# B&R Automation Studio project A2019059_Linka_Power_CP (part 33)

```iecst
            IF P2_StoperZvarania.IN.Centrovanie_ZASUNUTE_IS17 THEN
                SC_P2_StoperZvarania.ResetStep:= TRUE;
                SC_P2_StoperZvarania.Step:= 550;
            END_IF

            //Odoslanie dát na server//

        550:
            SC_P2_StoperZvarania.StepName:='550 - Automaticky Rezim - odoslanie stavu paletky na server';
            SC_P2_StoperZvarania.IdleTime.PT:= T#200ms;
            SC_P2_StoperZvarania.AlarmTime.PT:= T#5s;

            IF NOT SC_P2_StoperZvarania.Switch1 THEN
                TRCB_P2_Zvaranie_ST6.CMD.OdosliStavPaletky_TYP2:= TRUE;
                SC_P2_StoperZvarania.Switch1:= TRUE;
            END_IF

            IF TRCB_P2_Zvaranie_ST6.STATUS.KomunikaciaUkoncena THEN
                TRCB_P2_Zvaranie_ST6.CMD.OdosliStavPaletky_TYP2:= FALSE;
                SC_P2_StoperZvarania.ResetStep:= TRUE;
                SC_P2_StoperZvarania.Step:= 553;
            ELSIF TRCB_P2_Zvaranie_ST6.STATUS.KomunikaciaError THEN
                //                P2_Alarmy[236]:= TRUE;
                //                P2_PoruchaST4:= TRUE;
            END_IF

        553:
            SC_P2_StoperZvarania.StepName:='553 - Automaticky Rezim - kontrola odpovede servera';
            SC_P2_StoperZvarania.IdleTime.PT:= T#200ms;
            SC_P2_StoperZvarania.AlarmTime.PT:= T#5s;

            IF NOT TRCB_P2_Zvaranie_ST6.STATUS.KomunikaciaUkoncena THEN
                IF TRCB_P2_Zvaranie_ST6.OUTPUTS.PovolenieCinnostiNaPaletke = 'OK' THEN
                    SC_P2_StoperZvarania.ResetStep:= TRUE;
                    SC_P2_StoperZvarania.Step:= 555;
                ELSIF TRCB_P2_Zvaranie_ST6.OUTPUTS.PovolenieCinnostiNaPaletke = 'NG' THEN
                    Paletka[i].PAR.StavPaletky:= 'NG';
                    SC_P2_StoperZvarania.ResetStep:= TRUE;
                    SC_P2_StoperZvarania.Step:= 555;
                END_IF
            END_IF

        555:
            SC_P2_StoperZvarania.StepName:='555 - Automaticky Rezim - vyhodnotenie stavu paletky';
            SC_P2_StoperZvarania.IdleTime.PT:= T#200ms;
            SC_P2_StoperZvarania.AlarmTime.PT:= T#10s;

            IF Paletka[i].PAR.StavPaletky = 'OK' THEN
                IF Paletka[i].PAR.StavPowerCP = 'PASS' THEN
                    Paletka[i].PAR.StavPaletky:= 'OK';
                ELSIF Paletka[i].PAR.StavPowerCP = 'FAIL' THEN
                    Paletka[i].PAR.StavPaletky:= 'NG';
                END_IF
            END_IF
            Paletka[i].VnutornyStav.KomunikaciaUzavreta:= TRUE;
            SC_P2_StoperZvarania.ResetStep:= TRUE;
            SC_P2_StoperZvarania.Step:= 560;

            //Vyvezenie paletky//

        560:
            SC_P2_StoperZvarania.StepName:='560 - Automaticky Rezim - cakam na vyvezenie na vstupny stoper bunky 3';
            SC_P2_StoperZvarania.IdleTime.PT:= T#200ms;
            SC_P2_StoperZvarania.AlarmTime.PT:= T#5s;

            IF P2_StoperZvarania.KoniecCyklu THEN
                SC_P2_StoperZvarania.ResetStep:= TRUE;
                SC_P2_StoperZvarania.Step:= 0;
            ELSIF ((NOT P3_VstupnyStoper.IN.PritomnPaletky_IS85 AND SC_P3_VstupnyStoper.Step = 100) OR (P3_VstupnyStoper.OUT.ZasunStoper_YV193 AND SC_P3_VstupnyStoper.Step = 105)) AND NOT P2_StoperZvarania.STAV.PrebiehaVyvezeniePaletky AND NOT TEST THEN
                P2_StoperZvarania.OUT.ZasunStoper_YV59:= TRUE;
                P2_StoperZvarania.STAV.PrebiehaVyvezeniePaletky:= TRUE;
                SC_P2_StoperZvarania.ResetStep:= TRUE;
                SC_P2_StoperZvarania.Step:= 561;
            END_IF

        561:
            SC_P2_StoperZvarania.StepName:='561 - Automaticky Rezim - ukoncenie vyvazania na vstupny stoper bunky 3';
            SC_P2_StoperZvarania.IdleTime.PT:= T#200ms;
            SC_P2_StoperZvarania.AlarmTime.PT:= T#10s;

            SC_P2_StoperZvarania.AlarmTime.IN:= P2_StoperZvarania.IN.PritomnostPaletky_S9;
            SC_P2_StoperZvarania.IdleTime.IN:= NOT P2_StoperZvarania.IN.PritomnostPaletky_S9;

            IF NOT P2_StoperZvarania.IN.PritomnostPaletky_S9 THEN
                IF Revork THEN
                    Paletka[i].PAR.RevorkovyKus:= FALSE;
                    Paletka[i].PAR.CisloRevorkovejStanice:= '';
                    Revork:= FALSE;
                END_IF
                TestovaciKus:= FALSE;
                CisloFotky:= 0;
                Paletka[i].PAR.StavPowerCP:= '';
                Paletka[i].VnutornyStav.CinnostSpustena:= FALSE;
                Paletka[i].VnutornyStav.CinnostUkoncena:= FALSE;
                Paletka[i].VnutornyStav.FotkyOdoslane:= FALSE;
                Paletka[i].VnutornyStav.KomunikaciaOtvorena:= FALSE;
                Paletka[i].VnutornyStav.KomunikaciaUzavreta:= FALSE;
                Reports.Zvaranie.Moment.LavyZvar:= '';
                Reports.Zvaranie.VyslednyReport:= '';
                Reports.Zvaranie.Vyska.LavyZvar:= '';
                Reports.Zvaranie.Frekvencia:= '';
                Reports.Zvaranie.Moment.PravyZvar:= '';
                Reports.Zvaranie.Vyska.PravyZvar:= '';
                Reports.Kamery.P2_CAM11_KontrolaZvaru:= '';
                Reports.Kamery.P2_CAM11_KontrolaPowerCP:= '';
            END_IF

            IF SC_P2_StoperZvarania.IdleTime.Q THEN
                P2_StoperZvarania.OUT.ZasunStoper_YV59:= FALSE;
                SC_P2_StoperZvarania.ResetStep:= TRUE;
                SC_P2_StoperZvarania.Step:= 100;
            ELSIF SC_P2_StoperZvarania.AlarmTime.Q THEN
                P2_Alarmy[289]:= TRUE;
                P2_Pracovisko.KoniecCyklu:= TRUE;
                SC_P2_StoperZvarania.ResetStep:= TRUE;
                SC_P2_StoperZvarania.Step:= 0;
            END_IF

            //*******************************************************Manuálny režim*******************************************************************************//

        700:
            SC_P2_StoperZvarania.StepName:='700 - Manualny Rezim';
            SC_P2_StoperZvarania.IdleTime.PT:= T#8s;
            SC_P2_StoperZvarania.AlarmTime.PT:= T#5s;

    END_CASE

                END_PROGRAM

PROGRAM _EXIT
                (* Insert code here *)

                END_PROGRAM
```

#### Variables.var - Local variables
```iecst
VAR
	SC_OvlCentrovacky : SequenceControlTyp;
	Centrovacku_VYSUN : BOOL;
	Centrovacku_ZASUN : BOOL;
	PrecitaneCisloPaletky : STRING[3];
	ServerOdpoved_StavPowerCP : STRING[5];
	i : USINT;
	TEST : BOOL;
	PocetDopytovNaServer : USINT;
	TestovaciKus : BOOL;
	Revork : BOOL;
	Triger_0 : BOOL;
	Triger_1 : BOOL;
	CisloFotky : USINT;
	PocetZopakovaniOdobratia : USINT;
	PocetTrigrovKamery : USINT;
END_VAR
```

#### OvlCentrovacky.st
```iecst
ACTION OvlCentrovacky:

	//Volanie funkcie SequenceControl//
	SequenceControl(SC:= SC_OvlCentrovacky);

	CASE SC_OvlCentrovacky.Step OF

		0:
			SC_OvlCentrovacky.StepName:= '0 - Nulovanie';
			Centrovacku_VYSUN:= FALSE;
			Centrovacku_ZASUN:= FALSE;
//			P2_StoperZvarania.OUT.VysunCentrovanie_YV60:= FALSE;
//			P2_StoperZvarania.OUT.ZasunCentrovanie_YV61:= FALSE;

			IF SC_P2_StoperZvarania.Step <> 0 THEN
				SC_OvlCentrovacky.ResetStep:= TRUE;
				SC_OvlCentrovacky.Step:= 1;
			END_IF

		1:
			SC_OvlCentrovacky.StepName:= '1 - Rozhodnutie o cinnosti';
			IF Centrovacku_VYSUN THEN
				SC_OvlCentrovacky.Step:= 10;
			ELSIF Centrovacku_ZASUN THEN
				SC_OvlCentrovacky.Step:= 20;
			END_IF

		10:
			SC_OvlCentrovacky.StepName:= '10 - Vysunutie centrovacky';
			SC_OvlCentrovacky.IdleTime.PT:= T#3s;
			SC_OvlCentrovacky.AlarmTime.PT:= T#3s;

			IF P2_StoperZvarania.Automat THEN
				SC_OvlCentrovacky.AlarmTime.IN:= TRUE;
			ELSE
				SC_OvlCentrovacky.IdleTime.IN:= TRUE;
			END_IF

			IF NOT SC_OvlCentrovacky.Switch1 THEN
				P2_StoperZvarania.OUT.ZasunCentrovanie_YV61:= FALSE;
                P2_StoperZvarania.OUT.VysunCentrovanie_YV60:= TRUE;
				SC_OvlCentrovacky.Switch1:= TRUE;
			END_IF

			IF P2_StoperZvarania.IN.Centrovanie_VYSUNUTE_IS16 OR SC_OvlCentrovacky.IdleTime.Q THEN
				SC_OvlCentrovacky.ResetStep:= TRUE;
				SC_OvlCentrovacky.Step:= 0;
			ELSIF SC_OvlCentrovacky.AlarmTime.Q THEN
				P2_Alarmy[217]:= TRUE;
				P2_PoruchaST4:= TRUE;
			END_IF

		20:
			SC_OvlCentrovacky.StepName:= '20 - Zasunutie centrovacky';
			SC_OvlCentrovacky.IdleTime.PT:= T#3s;
			SC_OvlCentrovacky.AlarmTime.PT:= T#3s;

			IF P2_StoperZvarania.Automat THEN
				SC_OvlCentrovacky.AlarmTime.IN:= TRUE;
			ELSE
				SC_OvlCentrovacky.IdleTime.IN:= TRUE;
			END_IF

			IF NOT SC_OvlCentrovacky.Switch1 THEN
				P2_StoperZvarania.OUT.VysunCentrovanie_YV60:= FALSE;
                P2_StoperZvarania.OUT.ZasunCentrovanie_YV61:= TRUE;
				SC_OvlCentrovacky.Switch1:= TRUE;
			END_IF

			IF P2_StoperZvarania.IN.Centrovanie_ZASUNUTE_IS17 OR SC_OvlCentrovacky.IdleTime.Q THEN
				SC_OvlCentrovacky.ResetStep:= TRUE;
				SC_OvlCentrovacky.Step:= 0;
			ELSIF SC_OvlCentrovacky.AlarmTime.Q THEN
				P2_Alarmy[218]:= TRUE;
				P2_PoruchaST4:= TRUE;
			END_IF

	END_CASE

END_ACTION
```

#### StratoveSekundy.st
```iecst
ACTION StratoveSekundy:

END_ACTION
```

#### IOLinkKomunikacia.st
```iecst
ACTION IOLinkKomunikacia:

	//Snímač paletky//
	P2_StoperZvarania.IN.PritomnostPaletky_S9:= P2_StoperZvarania.PAR.SnimacPaletky_IOLinkInputs[1].0;
	P2_StoperZvarania.IN.PrecitaneCisloPaletky_S9:= P2_StoperZvarania.PAR.SnimacPaletky_IOLinkInputs[9];

END_ACTION
```

### Program Logical/Program/Pracovisko_2/P2_Zvaranie (IEC)

#### Main.st - Init, cyclic, exit code
```iecst
PROGRAM _INIT
    P2_Zvaranie.PAR.ServoZdvihu_JoggRychlost:= 5;

    //Zápis do ParID serva - nastavenie max momentu v smere otáčania a v protismere otáčania//
//    NovaHodnotaMomentu_POS := 1.5; //v Nm
//    NovaHodnotaMomentu_NEG := 1.5; //v Nm
//    MC_BR_ProcessParID_AcpAx_0.Axis:= ADR(gAxis_5);
//    MC_BR_ProcessParID_AcpAx_0.DataAddress:= ADR(McAcpAxProcessParIDType_0);
//    MC_BR_ProcessParID_AcpAx_0.NumberOfParIDs:= 2;
//    MC_BR_ProcessParID_AcpAx_0.Mode:= mcACPAX_PARID_SET;
//
//    McAcpAxProcessParIDType_0[0].DataType   := mcACPAX_PARTYPE_REAL;
//    McAcpAxProcessParIDType_0[0].ParID      := 248;
//    McAcpAxProcessParIDType_0[0].VariableAddress    := ADR(NovaHodnotaMomentu_POS);
//
//    McAcpAxProcessParIDType_0[1].DataType   := mcACPAX_PARTYPE_REAL;
//    McAcpAxProcessParIDType_0[1].ParID      := 249;
//    McAcpAxProcessParIDType_0[1].VariableAddress    := ADR(NovaHodnotaMomentu_NEG);
//
//    MC_BR_ProcessParID_AcpAx_0.Execute:= TRUE;
//    MC_BR_ProcessParID_AcpAx_0();

END_PROGRAM

PROGRAM _CYCLIC

     //Index paletky//
    i:= P2_StoperZvarania.PAR.IndexPaletky;

    //Volanie funkcie SequenceControl//
    SequenceControl(SC:= SC_P2_Zvaranie);

    //Volanie podprogramov//
    OvlServaZdvihu;
    OvlPojazdu;

    //Reset sekcie //
    IF NOT Safety.STAV.P2_ZonaBunky_AKTIVNA THEN
        SC_P2_Zvaranie.Step:= 0;
    ELSIF P2_Zvaranie.Reset THEN
        SC_P2_Zvaranie.Step:= 0;
        P2_Zvaranie.Reset:= FALSE;
    END_IF

    //Zastavenie serva//
    IF EDGEPOS(P2_PoruchaST4) THEN
        Zdvih_STOP:= TRUE;
    ELSIF EDGEPOS(P2_Zvaranie.Reset) THEN
        Zdvih_STOP:= TRUE;
    END_IF

    CASE SC_P2_Zvaranie.Step OF

        0:
            SC_P2_Zvaranie.StepName:='0 - Nulovanie';
            SC_OvlZdvihu.Step:= 0;
            P2_Zvaranie.Automat:= FALSE;
            P2_Zvaranie.KoniecCyklu:= FALSE;
            P2_Zvaranie.Manual:= FALSE;
            P2_Zvaranie.STAV.PoINIT:= FALSE;
            P2_Zvaranie.ServoZdvihuZvarania_M6.CMD.JoggLimit_ACTIVE:= FALSE;
            P2_Robot.KOM_OUT.Zvaranie_BezpecnaPozicia:= FALSE;
            P2_Zvaranie.STAV.ServoZdvihu_PoziciaDosiahnuta:= FALSE;
            P2_Zvaranie.OUT.Zvaracka_RESET:= FALSE;
            P2_Zvaranie.OUT.Zvaracka_START:= FALSE;

            IF Safety.STAV.P2_ZonaBunky_AKTIVNA AND NOT P2_Pracovisko.STAV.PORUCHA AND P2_Pracovisko.IN.PrivodVzduchu_SnimacTlaku_S3 AND P2_Pracovisko.STAV.ServaBunky_READY THEN
                SC_P2_Zvaranie.ResetStep:= TRUE;
                SC_P2_Zvaranie.Step:= 1;
            END_IF

        1:
            SC_P2_Zvaranie.StepName:='1 - Cakam na spustenie vyroby';
            P2_Zvaranie.KoniecCyklu:= FALSE;
            IF P2_Zvaranie.Automat THEN
                SC_P2_Zvaranie.Step:= 2;
            ELSIF P2_Zvaranie.Manual THEN
                SC_P2_Zvaranie.Step:= 700;
            END_IF

            //********************************************************Inicializácia****************************************************************************//

        2:
            SC_P2_Zvaranie.StepName:='2 - Inicializacia - cakam na spustenie inicializacie';
            SC_P2_Zvaranie.IdleTime.PT:= T#2s;
            SC_P2_Zvaranie.AlarmTime.PT:= T#5s;

            SC_P2_Zvaranie.IdleTime.IN:= TRUE;

            IF SC_P2_Zvaranie.IdleTime.Q THEN
                SC_P2_Zvaranie.ResetStep:= TRUE;
                SC_P2_Zvaranie.Step:= 3;
            END_IF

        3:
            SC_P2_Zvaranie.StepName:='3 - Inicializacia - kontrola homingu serva zdvihu zvarania';
            SC_P2_Zvaranie.IdleTime.PT:= T#2s;
            SC_P2_Zvaranie.AlarmTime.PT:= T#5s;

            IF P2_Zvaranie.STAV.ServoZdvihu_HomingOK THEN
                SC_P2_Zvaranie.ResetStep:= TRUE;
                SC_P2_Zvaranie.Step:= 5;
            ELSE
                SC_P2_Zvaranie.ResetStep:= TRUE;
                SC_P2_Zvaranie.Step:= 4;
            END_IF

        4:
            SC_P2_Zvaranie.StepName:='4 - Inicializacia - spustenie homingu serva zdvihu zvarania';
            SC_P2_Zvaranie.IdleTime.PT:= T#2s;
            SC_P2_Zvaranie.AlarmTime.PT:= T#5s;

            IF NOT SC_P2_Zvaranie.Switch1 AND Safety.STAV.P2_ZonaBunky_AKTIVNA THEN
                Zdvih_HOME:= TRUE;
                SC_P2_Zvaranie.Switch1:= TRUE;
            END_IF

            IF P2_Zvaranie.STAV.ServoZdvihu_HomingOK THEN
                SC_P2_Zvaranie.ResetStep:= TRUE;
                SC_P2_Zvaranie.Step:= 5;
            END_IF

        5:
            SC_P2_Zvaranie.StepName:='5 - Inicializacia - presun zdvihu zvarania do vychodiskovej pozicie';
            SC_P2_Zvaranie.IdleTime.PT:= T#2s;
            SC_P2_Zvaranie.AlarmTime.PT:= T#5s;

            P2_Zvaranie.PAR.ServoZdvihu_ZadanaPozicia:= 0;

            P2_Robot.KOM_OUT.Zvaranie_BezpecnaPozicia:= FALSE;

            IF NOT SC_P2_Zvaranie.Switch1 AND SC_OvlZdvihu.Step = 1 AND Safety.STAV.P2_ZonaBunky_AKTIVNA THEN
                Zdvih_POLOHUJ:= TRUE;
                SC_P2_Zvaranie.Switch1:= TRUE;
            END_IF

            IF P2_Zvaranie.STAV.ServoZdvihu_PoziciaDosiahnuta THEN
                P2_Zvaranie.STAV.ServoZdvihu_PoziciaDosiahnuta:= FALSE;
                SC_P2_Zvaranie.ResetStep:= TRUE;
                SC_P2_Zvaranie.Step:= 10;
            END_IF

        10:
            SC_P2_Zvaranie.StepName:='10 - Inicializacia - presun pojazdu zvarania vpravo';
            SC_P2_Zvaranie.IdleTime.PT:= T#2s;
            SC_P2_Zvaranie.AlarmTime.PT:= T#5s;

            IF NOT SC_P2_Zvaranie.Switch1 THEN
                PresunVPRAVO:= TRUE;
                SC_P2_Zvaranie.Switch1:= TRUE;
            END_IF

            IF P2_Zvaranie.IN.PojazdZvarania_PozVPRAVO_IS10 THEN
                P2_Robot.KOM_OUT.Zvaranie_BezpecnaPozicia:= TRUE;
                SC_P2_Zvaranie.ResetStep:= TRUE;
                SC_P2_Zvaranie.Step:= 12;
            END_IF

        12:
            SC_P2_Zvaranie.StepName:='12 - Inicializacia - kontrola stavu zvaracky';
            SC_P2_Zvaranie.IdleTime.PT:= T#2s;
            SC_P2_Zvaranie.AlarmTime.PT:= T#5s;

            IF NOT P2_Zvaranie.IN.ZvarackaStav_READY THEN
                SC_P2_Zvaranie.ResetStep:= TRUE;
                SC_P2_Zvaranie.Step:= 15;
            ELSE
                P2_Zvaranie.STAV.PoINIT:= TRUE;
                SC_P2_Zvaranie.ResetStep:= TRUE;
                SC_P2_Zvaranie.Step:= 100;
            END_IF

        15:
            SC_P2_Zvaranie.StepName:='15 - Inicializacia - reset zvaracky';
            SC_P2_Zvaranie.IdleTime.PT:= T#200ms;
            SC_P2_Zvaranie.AlarmTime.PT:= T#5s;

            IF NOT SC_P2_Zvaranie.Switch1 THEN
                P2_Zvaranie.OUT.Zvaracka_RESET:= TRUE;
                SC_P2_Zvaranie.IdleTime.IN:= TRUE;
                SC_P2_Zvaranie.Switch1:= TRUE;
            END_IF

            IF SC_P2_Zvaranie.IdleTime.Q THEN
                P2_Zvaranie.OUT.Zvaracka_RESET:= FALSE;
            END_IF

            IF P2_Zvaranie.IN.ZvarackaStav_READY THEN
                P2_Zvaranie.STAV.PoINIT:= TRUE;
                SC_P2_Zvaranie.ResetStep:= TRUE;
                SC_P2_Zvaranie.Step:= 100;
            END_IF

            //********************************************************Automatický režim****************************************************************************//

        100:
            SC_P2_Zvaranie.StepName:='100 - Automaticky Rezim - cakam na spustenie zvarania';
            SC_P2_Zvaranie.IdleTime.PT:= T#200ms;
            SC_P2_Zvaranie.AlarmTime.PT:= T#5s;

            P2_Robot.KOM_OUT.Zvaranie_BezpecnaPozicia:= TRUE;

            IF P2_Zvaranie.KoniecCyklu AND NOT P2_StoperZvarania.Automat THEN
                SC_P2_Zvaranie.ResetStep:= TRUE;
                SC_P2_Zvaranie.Step:= 0;
            ELSIF P2_StoperZvarania.OUT.KOM_Zvaranie_START THEN
                P2_Robot.KOM_OUT.Zvaranie_BezpecnaPozicia:= FALSE;
                SC_P2_Zvaranie.ResetStep:= TRUE;
                SC_P2_Zvaranie.Step:= 102;
            ELSIF  P2_StoperZvarania.OUT.KOM_Zatlacanie_START THEN
                P2_Robot.KOM_OUT.Zvaranie_BezpecnaPozicia:= FALSE;
                SC_P2_Zvaranie.ResetStep:= TRUE;
                SC_P2_Zvaranie.Step:= 200;
            END_IF

        102:
            SC_P2_Zvaranie.StepName:='102 - Automaticky Rezim - napolohovanie zdvihu zvaracky nad bod zvarania';
            SC_P2_Zvaranie.IdleTime.PT:= T#200ms;
            SC_P2_Zvaranie.AlarmTime.PT:= T#5s;

            P2_Zvaranie.PAR.ServoZdvihu_ZadanaPozicia:= 234;//240

            IF NOT SC_P2_Zvaranie.Switch1 AND SC_OvlZdvihu.Step = 1 AND Safety.STAV.P2_ZonaBunky_AKTIVNA THEN
                Zdvih_POLOHUJ:= TRUE;
                SC_P2_Zvaranie.Switch1:= TRUE;
            END_IF

            IF P2_Zvaranie.STAV.ServoZdvihu_PoziciaDosiahnuta THEN
                P2_Zvaranie.STAV.ServoZdvihu_PoziciaDosiahnuta:= FALSE;
                SC_P2_Zvaranie.ResetStep:= TRUE;
                SC_P2_Zvaranie.Step:= 105;
            END_IF

        105:
            SC_P2_Zvaranie.StepName:='105 - Automaticky Rezim - spustenie zvaracky';
            SC_P2_Zvaranie.IdleTime.PT:= T#500ms;
            SC_P2_Zvaranie.AlarmTime.PT:= T#2s;

            SC_P2_Zvaranie.AlarmTime.IN:= NOT P2_Zvaranie.IN.ZvarackaStav_READY;

            IF NOT SC_P2_Zvaranie.Switch1 AND P2_Zvaranie.IN.ZvarackaStav_READY THEN
                P2_Zvaranie.OUT.Zvaracka_START:= TRUE;
                SC_P2_Zvaranie.Switch1:= TRUE;
            END_IF

            IF P2_Zvaranie.IN.ZvarackaStav_RUN THEN
                SC_P2_Zvaranie.ResetStep:= TRUE;
                SC_P2_Zvaranie.Step:= 108;
            ELSIF SC_P2_Zvaranie.AlarmTime.Q THEN
                SC_P2_Zvaranie.ResetStep:= TRUE;
                SC_P2_Zvaranie.Step:= 106;
            END_IF

        106:
            SC_P2_Zvaranie.StepName:='106 - Automaticky Rezim - resetovanie zvaracky';
            SC_P2_Zvaranie.IdleTime.PT:= T#500ms;
            SC_P2_Zvaranie.AlarmTime.PT:= T#5s;

            IF NOT SC_P2_Zvaranie.Switch1 THEN
                P2_Zvaranie.OUT.Zvaracka_RESET:= TRUE;
                SC_P2_Zvaranie.IdleTime.IN:= TRUE;
                SC_P2_Zvaranie.Switch1:= TRUE;
            END_IF

            IF SC_P2_Zvaranie.IdleTime.Q THEN
                P2_Zvaranie.OUT.Zvaracka_RESET:= FALSE;
                SC_P2_Zvaranie.ResetStep:= TRUE;
                SC_P2_Zvaranie.Step:= 105;
            END_IF

        108:
            SC_P2_Zvaranie.StepName:='108 - Automaticky Rezim - zvaranie pravej casti';
            SC_P2_Zvaranie.IdleTime.PT:= T#200ms;
            SC_P2_Zvaranie.AlarmTime.PT:= T#5s;

            P2_Zvaranie.PAR.ServoZdvihu_ZadanyMoment:= P2_RemPremenne.P2_Zvaranie_MomentZvarania;

            IF NOT SC_P2_Zvaranie.Switch1 AND SC_OvlZdvihu.Step = 1 AND Safety.STAV.P2_ZonaBunky_AKTIVNA THEN
                Zdvih_ZVARANIE:= TRUE;
                SC_P2_Zvaranie.Switch1:= TRUE;
            END_IF

            IF P2_Zvaranie.STAV.ServoZdvihu_PoziciaDosiahnuta THEN
                P2_Zvaranie.STAV.ServoZdvihu_PoziciaDosiahnuta:= FALSE;
                Reports.Zvaranie.Moment.PravyZvar:= REAL_TO_STRING(P2_Zvaranie.ServoZdvihuZvarania_M6.STATUS.ActualTorque);
                Reports.Zvaranie.Vyska.PravyZvar:= LREAL_TO_STRING(P2_Zvaranie.STAV.Zdvih_AktualnaPozicia);
                Reports.Zvaranie.Frekvencia:= '80';
                P2_Zvaranie.STAV.Vysledok_Zvarania:= 'OK';
                SC_P2_Zvaranie.ResetStep:= TRUE;
                SC_P2_Zvaranie.Step:= 110;
            END_IF

//Zváranie//
        110:
            SC_P2_Zvaranie.StepName:='110 - Automaticky Rezim - napolohovanie zdvihu zvaracky nad bod zvarania, vypnutie zvaracky';
            SC_P2_Zvaranie.IdleTime.PT:= T#200ms;
            SC_P2_Zvaranie.AlarmTime.PT:= T#5s;

            P2_Zvaranie.PAR.ServoZdvihu_ZadanaPozicia:= 234;//240

            IF NOT SC_P2_Zvaranie.Switch1 AND SC_OvlZdvihu.Step = 1 AND Safety.STAV.P2_ZonaBunky_AKTIVNA THEN
                Zdvih_POLOHUJ:= TRUE;
                P2_Zvaranie.OUT.Zvaracka_START:= FALSE;
                SC_P2_Zvaranie.Switch1:= TRUE;
            END_IF

            IF P2_Zvaranie.STAV.ServoZdvihu_PoziciaDosiahnuta THEN
                P2_Zvaranie.STAV.ServoZdvihu_PoziciaDosiahnuta:= FALSE;
                SC_P2_Zvaranie.ResetStep:= TRUE;
                SC_P2_Zvaranie.Step:= 112;
            END_IF

        112:
            SC_P2_Zvaranie.StepName:='112 - Automaticky Rezim - presun pojazdu zvarania vlavo';
            SC_P2_Zvaranie.IdleTime.PT:= T#200ms;
            SC_P2_Zvaranie.AlarmTime.PT:= T#5s;

            IF NOT SC_P2_Zvaranie.Switch1 THEN
                PresunVLAVO:= TRUE;
                SC_P2_Zvaranie.Switch1:= TRUE;
            END_IF

            IF P2_Zvaranie.IN.PojazdZvarania_PozVLAVO_IS11 THEN
                SC_P2_Zvaranie.ResetStep:= TRUE;
                SC_P2_Zvaranie.Step:= 115;
            END_IF

        115:
            SC_P2_Zvaranie.StepName:='115 - Automaticky Rezim - spustenie zvaracky';
            SC_P2_Zvaranie.IdleTime.PT:= T#200ms;
            SC_P2_Zvaranie.AlarmTime.PT:= T#2s;

            SC_P2_Zvaranie.AlarmTime.IN:= NOT P2_Zvaranie.IN.ZvarackaStav_READY;

            IF NOT SC_P2_Zvaranie.Switch1 AND P2_Zvaranie.IN.ZvarackaStav_READY THEN
                P2_Zvaranie.OUT.Zvaracka_START:= TRUE;
                SC_P2_Zvaranie.Switch1:= TRUE;
            END_IF

            IF P2_Zvaranie.IN.ZvarackaStav_RUN THEN
                SC_P2_Zvaranie.ResetStep:= TRUE;
                SC_P2_Zvaranie.Step:= 118;
            ELSIF SC_P2_Zvaranie.AlarmTime.Q THEN
                SC_P2_Zvaranie.ResetStep:= TRUE;
                SC_P2_Zvaranie.Step:= 116;
            END_IF

        116:
            SC_P2_Zvaranie.StepName:='116 - Automaticky Rezim - resetovanie zvaracky';
            SC_P2_Zvaranie.IdleTime.PT:= T#500ms;
            SC_P2_Zvaranie.AlarmTime.PT:= T#5s;

            IF NOT SC_P2_Zvaranie.Switch1 THEN
                P2_Zvaranie.OUT.Zvaracka_RESET:= TRUE;
                SC_P2_Zvaranie.IdleTime.IN:= TRUE;
                SC_P2_Zvaranie.Switch1:= TRUE;
            END_IF

            IF SC_P2_Zvaranie.IdleTime.Q THEN
                P2_Zvaranie.OUT.Zvaracka_RESET:= FALSE;
                SC_P2_Zvaranie.ResetStep:= TRUE;
                SC_P2_Zvaranie.Step:= 115;
            END_IF

        118:
            SC_P2_Zvaranie.StepName:='118 - Automaticky Rezim - zvaranie lavej casti';
            SC_P2_Zvaranie.IdleTime.PT:= T#200ms;
            SC_P2_Zvaranie.AlarmTime.PT:= T#5s;

            IF NOT SC_P2_Zvaranie.Switch1 AND SC_OvlZdvihu.Step = 1 AND Safety.STAV.P2_ZonaBunky_AKTIVNA THEN
                Zdvih_ZVARANIE:= TRUE;
                SC_P2_Zvaranie.Switch1:= TRUE;
            END_IF

            IF P2_Zvaranie.STAV.ServoZdvihu_PoziciaDosiahnuta THEN
                P2_Zvaranie.STAV.ServoZdvihu_PoziciaDosiahnuta:= FALSE;
                P2_Zvaranie.STAV.Vysledok_Zvarania:= 'OK';
                Reports.Zvaranie.Moment.LavyZvar:= REAL_TO_STRING(P2_Zvaranie.ServoZdvihuZvarania_M6.STATUS.ActualTorque);
                Reports.Zvaranie.Vyska.LavyZvar:= LREAL_TO_STRING(P2_Zvaranie.STAV.Zdvih_AktualnaPozicia);
                Reports.Zvaranie.Frekvencia:= '80';
                SC_P2_Zvaranie.ResetStep:= TRUE;
                SC_P2_Zvaranie.Step:= 120;
            END_IF

        120:
            SC_P2_Zvaranie.StepName:='120 - Automaticky Rezim - napolohovanie zdvihu zvaracky do vychodiskovej polohy,presun vpravo a vypnutie zvaracky';
            SC_P2_Zvaranie.IdleTime.PT:= T#200ms;
            SC_P2_Zvaranie.AlarmTime.PT:= T#5s;

            P2_Zvaranie.PAR.ServoZdvihu_ZadanaPozicia:= 0;

            IF NOT SC_P2_Zvaranie.Switch1 AND SC_OvlZdvihu.Step = 1 AND Safety.STAV.P2_ZonaBunky_AKTIVNA THEN
                Zdvih_POLOHUJ:= TRUE;
                P2_Zvaranie.OUT.Zvaracka_START:= FALSE;
                SC_P2_Zvaranie.Switch1:= TRUE;
            END_IF

            IF EDGEPOS(P2_Zvaranie.STAV.Zdvih_AktualnaPozicia < 200) THEN
                PresunVPRAVO:= TRUE;
            END_IF

            IF P2_Zvaranie.STAV.ServoZdvihu_PoziciaDosiahnuta AND P2_Zvaranie.IN.PojazdZvarania_PozVPRAVO_IS10 THEN
                P2_Zvaranie.STAV.ServoZdvihu_PoziciaDosiahnuta:= FALSE;
                SC_P2_Zvaranie.ResetStep:= TRUE;
                SC_P2_Zvaranie.Step:= 122;
            END_IF

        122:
            SC_P2_Zvaranie.StepName:='122 - Automaticky Rezim - vystavenie signalu ukoncenie zvarania';
            SC_P2_Zvaranie.IdleTime.PT:= T#200ms;
            SC_P2_Zvaranie.AlarmTime.PT:= T#5s;

            P2_Robot.KOM_OUT.Zvaranie_BezpecnaPozicia:= TRUE;

            IF NOT SC_P2_Zvaranie.Switch1 THEN
                P2_Zvaranie.OUT.KOM_ZavaranieUkoncene:= TRUE;
                SC_P2_Zvaranie.Switch1:= TRUE;
            END_IF

            IF NOT P2_StoperZvarania.OUT.KOM_Zvaranie_START THEN
                SC_P2_Zvaranie.ResetStep:= TRUE;
                SC_P2_Zvaranie.Step:= 100;
            END_IF

//Zatláčanie Coveru//

        200:
            SC_P2_Zvaranie.StepName:='200 - Automaticky Rezim - napolohovanie zdvihu zatlacania nad bod zatlacenia';
            SC_P2_Zvaranie.IdleTime.PT:= T#200ms;
            SC_P2_Zvaranie.AlarmTime.PT:= T#5s;

            P2_Zvaranie.PAR.ServoZdvihu_ZadanaPozicia:= 200;

            IF NOT SC_P2_Zvaranie.Switch1 THEN
                PresunVLAVO:= TRUE;
                SC_P2_Zvaranie.Switch1:= TRUE;
            END_IF

            IF NOT SC_P2_Zvaranie.Switch2 AND SC_OvlZdvihu.Step = 1 AND Safety.STAV.P2_ZonaBunky_AKTIVNA AND P2_Zvaranie.IN.PojazdZvarania_PozVLAVO_IS11 THEN
                Zdvih_POLOHUJ:= TRUE;
                SC_P2_Zvaranie.Switch2:= TRUE;
            END_IF

            IF P2_Zvaranie.STAV.ServoZdvihu_PoziciaDosiahnuta THEN
                P2_Zvaranie.STAV.ServoZdvihu_PoziciaDosiahnuta:= FALSE;
                SC_P2_Zvaranie.ResetStep:= TRUE;
                SC_P2_Zvaranie.Step:= 205;
            END_IF

        205:
            SC_P2_Zvaranie.StepName:='205 - Automaticky Rezim - zatlacanie coveru';
            SC_P2_Zvaranie.IdleTime.PT:= T#200ms;
            SC_P2_Zvaranie.AlarmTime.PT:= T#5s;

            IF NOT SC_P2_Zvaranie.Switch1 AND SC_OvlZdvihu.Step = 1 AND Safety.STAV.P2_ZonaBunky_AKTIVNA THEN
                Zdvih_ZATLACANIE:= TRUE;
                SC_P2_Zvaranie.Switch1:= TRUE;
            END_IF

            IF P2_Zvaranie.STAV.ServoZdvihu_PoziciaDosiahnuta THEN
                P2_Zvaranie.STAV.ServoZdvihu_PoziciaDosiahnuta:= FALSE;
                SC_P2_Zvaranie.ResetStep:= TRUE;
                SC_P2_Zvaranie.Step:= 208;
            END_IF

        208:
            SC_P2_Zvaranie.StepName:='208 - Automaticky Rezim - napolohovanie zdvihu zatlacania do vychodiskovej polohy';
            SC_P2_Zvaranie.IdleTime.PT:= T#200ms;
            SC_P2_Zvaranie.AlarmTime.PT:= T#5s;

            P2_Zvaranie.PAR.ServoZdvihu_ZadanaPozicia:= 0;

            IF NOT SC_P2_Zvaranie.Switch1 AND SC_OvlZdvihu.Step = 1 AND Safety.STAV.P2_ZonaBunky_AKTIVNA THEN
                Zdvih_POLOHUJ:= TRUE;
                SC_P2_Zvaranie.Switch1:= TRUE;
            END_IF

            IF EDGEPOS(P2_Zvaranie.STAV.Zdvih_AktualnaPozicia < 200) THEN
                PresunVPRAVO:= TRUE;
            END_IF

            IF P2_Zvaranie.STAV.ServoZdvihu_PoziciaDosiahnuta AND P2_Zvaranie.IN.PojazdZvarania_PozVPRAVO_IS10 THEN
                P2_Zvaranie.STAV.ServoZdvihu_PoziciaDosiahnuta:= FALSE;
                SC_P2_Zvaranie.ResetStep:= TRUE;
                SC_P2_Zvaranie.Step:= 210;
            END_IF

        210:
            SC_P2_Zvaranie.StepName:='210 - Automaticky Rezim - vystavenie signalu ukoncenie zatlacania';
            SC_P2_Zvaranie.IdleTime.PT:= T#200ms;
            SC_P2_Zvaranie.AlarmTime.PT:= T#5s;

            P2_Robot.KOM_OUT.Zvaranie_BezpecnaPozicia:= TRUE;

            IF NOT SC_P2_Zvaranie.Switch1 THEN
                P2_Zvaranie.OUT.KOM_ZatlacanieUkoncene:= TRUE;
                SC_P2_Zvaranie.Switch1:= TRUE;
            END_IF

            IF NOT P2_StoperZvarania.OUT.KOM_Zatlacanie_START THEN
                SC_P2_Zvaranie.ResetStep:= TRUE;
                SC_P2_Zvaranie.Step:= 100;
            END_IF

            //*******************************************************Manuálny režim*******************************************************************************//
        700:
            SC_P2_Zvaranie.StepName:='700 - Manualny Rezim';
            SC_P2_Zvaranie.IdleTime.PT:= T#8s;
            SC_P2_Zvaranie.AlarmTime.PT:= T#5s;

            P2_Zvaranie.ServoZdvihuZvarania_M6.PAR.JoggAcceleration:= (P2_Zvaranie.PAR.ServoZdvihu_JoggRychlost * 10);
            P2_Zvaranie.ServoZdvihuZvarania_M6.PAR.JoggDeceleration:= (P2_Zvaranie.PAR.ServoZdvihu_JoggRychlost * 10);
            P2_Zvaranie.ServoZdvihuZvarania_M6.PAR.JoggVelocity:= P2_Zvaranie.PAR.ServoZdvihu_JoggRychlost;
            P2_Zvaranie.ServoZdvihuZvarania_M6.PAR.JoggPoziciaLimitVPRED:= 250.0;
            P2_Zvaranie.ServoZdvihuZvarania_M6.PAR.JoggPoziciaLimitVZAD:= 0.0;
            P2_Zvaranie.ServoZdvihuZvarania_M6.CMD.JoggLimit_ACTIVE:= TRUE;

    END_CASE

END_PROGRAM

PROGRAM _EXIT
	(* Insert code here *)

END_PROGRAM
```

#### Variables.var - Local variables
```iecst
VAR
	SC_OvlZvarania : SequenceControlTyp;
	PocetBlikovREADY : USINT;
	SC_OvlZdvihu : SequenceControlTyp;
	Zdvih_JoggDOLE : BOOL;
	Zdvih_JoggHORE : BOOL;
	Zdvih_POLOHUJ : BOOL;
	Zdvih_HOME : BOOL;
	Zdvih_STOP : BOOL;
	Zdvih_ZVARANIE : BOOL;
	Zdvih_ZATLACANIE : BOOL;
	SC_OvlPojazdu : SequenceControlTyp;
	PresunVPRAVO : BOOL;
	PresunVLAVO : BOOL;
END_VAR
VAR RETAIN
	CasZotrvaniaZvarania : TIME;
	TorqRychlost : REAL;
	TorqMoment : REAL;
END_VAR
VAR
	ZadanaPoziciaUINT : UINT;
	AktualnaPoziciaUINT : UINT;
	MomentDosiahnuty : BOOL;
	CasPowerON : TON;
	i : USINT;
	CasZastaveniaServa : TON;
END_VAR
(******Zápis do ParID serva*************)
VAR
	MC_BR_ProcessParID_AcpAx_0 : MC_BR_ProcessParID_AcpAx := (0);
	McAcpAxProcessParIDType_0 : ARRAY[0..1] OF McAcpAxProcessParIDType;
	NovaHodnotaMomentu_POS : REAL := 0.0;
	NovaHodnotaMomentu_NEG : REAL := 0.0;
END_VAR
```

#### OvlServaZdvihu.st
```iecst
ACTION OvlServaZdvihu:

	//**************************Axis 5***********************************//
	//Otáčka serva = 10mm//
	//Motor má absolútny encodér a brzdu//

    //ENABLE knižnice//
    IF P2_Zvaranie.ServoZdvihuZvarania_M6.STATUS.Communication_READY THEN
        P2_Zvaranie.ServoZdvihuZvarania_M6.CMD.ENABLE:= TRUE;
    ELSE
        P2_Zvaranie.ServoZdvihuZvarania_M6.CMD.ENABLE:= FALSE;
    END_IF

	//Zapnutie serva//
	CasPowerON.IN:= P2_Zvaranie.ServoZdvihuZvarania_M6.STATUS.ReadyToPower_ON AND P2_Zvaranie.STAV.ServoZvihu_LimitSnimace_BUSY AND P2_Zvaranie.ServoZdvihuZvarania_M6.STATUS.EnableSwitch_ACTIVE AND NOT P2_Zvaranie.ServoZdvihuZvarania_M6.STATUS.ERROR;
	IF CasPowerON.Q THEN
		P2_Zvaranie.ServoZdvihuZvarania_M6.CMD.POWER:= TRUE;
	ELSE
		P2_Zvaranie.ServoZdvihuZvarania_M6.CMD.POWER:= FALSE;
	END_IF

	CasPowerON.PT:= T#1s;
	CasPowerON();

    //Zobrazenie stavou a parametrov serva//
    P2_Zvaranie.STAV.Zdvih_AktualnaPozicia:= P2_Zvaranie.ServoZdvihuZvarania_M6.STATUS.ActualPosition;
	P2_Zvaranie.STAV.Zdvih_AktualnaRychlost:= P2_Zvaranie.ServoZdvihuZvarania_M6.STATUS.ActualVelocity;
	P2_Zvaranie.STAV.Zdvih_AktualnyMoment:= P2_Zvaranie.ServoZdvihuZvarania_M6.STATUS.ActualTorque;
	P2_Zvaranie.STAV.ServoZdvihu_HomingOK:= P2_Zvaranie.ServoZdvihuZvarania_M6.STATUS.Homing_OK;
	P2_Zvaranie.STAV.ServoZdvihu_BUSY:= P2_Zvaranie.ServoZdvihuZvarania_M6.STATUS.MoveAbsolute_BUSY;
	P2_Zvaranie.STAV.Zdvih_JoggLimitDosiahnuty:= P2_Zvaranie.ServoZdvihuZvarania_M6.STATUS.JoggLimit_Dosiahnuty;

	//Zadané parametre serva//
	P2_Zvaranie.ServoZdvihuZvarania_M6.HomePAR.Acceleration:= 100;
	P2_Zvaranie.ServoZdvihuZvarania_M6.HomePAR.HomingVelocity:= 5;
	P2_Zvaranie.ServoZdvihuZvarania_M6.HomePAR.StartVelocity:= 10;
	P2_Zvaranie.ServoZdvihuZvarania_M6.HomePAR.Position:= -37731.5;    //Offset homing pozície pre absolutny snímač
	P2_Zvaranie.ServoZdvihuZvarania_M6.HomePAR.HomingMode:= 3; //0 - direct, 1- refrenčný snímač, 2 - limitný snímač, 3 - absolutny encoder, 4 - na moment//

	P2_Zvaranie.ServoZdvihuZvarania_M6.PAR.Acceleration:= P2_RemPremenne.P2_ZdvihZvarania_Rychlost*10;
	P2_Zvaranie.ServoZdvihuZvarania_M6.PAR.Deceleration:= P2_RemPremenne.P2_ZdvihZvarania_Rychlost*10;
	P2_Zvaranie.ServoZdvihuZvarania_M6.PAR.StopDeceleration:= P2_RemPremenne.P2_ZdvihZvarania_Rychlost*10;
	P2_Zvaranie.ServoZdvihuZvarania_M6.PAR.Velocity:= P2_RemPremenne.P2_ZdvihZvarania_Rychlost;
    P2_Zvaranie.ServoZdvihuZvarania_M6.PAR.Position:= P2_Zvaranie.PAR.ServoZdvihu_ZadanaPozicia;

    //Zastavenie pohybu serva//
	IF Zdvih_STOP THEN
		P2_Zvaranie.ServoZdvihuZvarania_M6.CMD.STOP:= TRUE;
		SC_OvlZdvihu.Step:= 0;
		CasZastaveniaServa.IN:= TRUE;
		Zdvih_STOP:= FALSE;
	END_IF

	IF CasZastaveniaServa.Q THEN
		P2_Zvaranie.ServoZdvihuZvarania_M6.CMD.STOP:= FALSE;
		CasZastaveniaServa.IN:= FALSE;
	END_IF

	CasZastaveniaServa.PT:= T#2s;
	CasZastaveniaServa();

	//Volanie funkcie SequenceControl//
	SequenceControl(SC:= SC_OvlZdvihu);

	CASE SC_OvlZdvihu.Step OF

		0:
			SC_OvlZdvihu.StepName:= '0 - Nulovanie';
			Zdvih_JoggHORE:= FALSE;
			Zdvih_JoggDOLE:= FALSE;
			Zdvih_POLOHUJ:= FALSE;
			Zdvih_HOME:= FALSE;
            Zdvih_ZVARANIE:= FALSE;
            Zdvih_ZATLACANIE:= FALSE;
			P2_Zvaranie.ServoZdvihuZvarania_M6.CMD.HOME:= FALSE;
			P2_Zvaranie.ServoZdvihuZvarania_M6.CMD.JoggVPRED:= FALSE;
			P2_Zvaranie.ServoZdvihuZvarania_M6.CMD.JoggVZAD:= FALSE;
			P2_Zvaranie.ServoZdvihuZvarania_M6.CMD.MoveAbsolute:= FALSE;
			P2_Zvaranie.ServoZdvihuZvarania_M6.CMD.MoveTorque:= FALSE;
			MomentDosiahnuty:= FALSE;

			IF SC_P2_Zvaranie.Step <> 0 AND P2_Zvaranie.ServoZdvihuZvarania_M6.STATUS.Power_ON AND NOT P2_Zvaranie.ServoZdvihuZvarania_M6.STATUS.ERROR AND NOT P2_Zvaranie.ServoZdvihuZvarania_M6.STATUS.STOP_ACTIVE THEN
				SC_OvlZdvihu.ResetStep:= TRUE;
				SC_OvlZdvihu.Step:= 1;
			END_IF

		1:
			SC_OvlZdvihu.StepName:= '1 - Rozhodnutie o cinnosti';
			IF Zdvih_JoggHORE THEN
				SC_OvlZdvihu.Step:= 10;
			ELSIF Zdvih_JoggDOLE THEN
				SC_OvlZdvihu.Step:= 20;
			ELSIF Zdvih_HOME THEN
				SC_OvlZdvihu.Step:= 30;
			ELSIF Zdvih_POLOHUJ THEN
				SC_OvlZdvihu.Step:= 40;
			ELSIF Zdvih_ZVARANIE THEN
                SC_OvlZdvihu.Step:= 50;
            ELSIF Zdvih_ZATLACANIE THEN
                SC_OvlZdvihu.Step:= 60;
			END_IF

		10:
			SC_OvlZdvihu.StepName:= '10 - Jogg HORE';
			SC_OvlZdvihu.IdleTime.PT:= T#3s;
			SC_OvlZdvihu.AlarmTime.PT:= T#3s;

			IF NOT SC_OvlZdvihu.Switch1 THEN
				P2_Zvaranie.ServoZdvihuZvarania_M6.CMD.JoggVZAD:= TRUE;
				SC_OvlZdvihu.Switch1:= TRUE;
			END_IF

			IF NOT Zdvih_JoggHORE THEN
				SC_OvlZdvihu.ResetStep:= TRUE;
				SC_OvlZdvihu.Step:= 0;
			END_IF

		20:
			SC_OvlZdvihu.StepName:= '20 - Jogg DOLE';
			SC_OvlZdvihu.IdleTime.PT:= T#3s;
			SC_OvlZdvihu.AlarmTime.PT:= T#3s;

			IF NOT SC_OvlZdvihu.Switch1 THEN
				P2_Zvaranie.ServoZdvihuZvarania_M6.CMD.JoggVPRED:= TRUE;
				SC_OvlZdvihu.Switch1:= TRUE;
			END_IF

			IF NOT Zdvih_JoggDOLE THEN
				SC_OvlZdvihu.ResetStep:= TRUE;
				SC_OvlZdvihu.Step:= 0;
			END_IF

		30:
			SC_OvlZdvihu.StepName:= '30 - Homing';
			SC_OvlZdvihu.IdleTime.PT:= T#500ms;
			SC_OvlZdvihu.AlarmTime.PT:= T#3s;

			IF NOT SC_OvlZdvihu.Switch1 THEN
				P2_Zvaranie.ServoZdvihuZvarania_M6.CMD.HOME:= TRUE;
				SC_OvlZdvihu.IdleTime.IN:= TRUE;
				SC_OvlZdvihu.Switch1:= TRUE;
			END_IF

			IF P2_Zvaranie.ServoZdvihuZvarania_M6.STATUS.Homing_OK AND SC_OvlZdvihu.IdleTime.Q THEN
				SC_OvlZdvihu.ResetStep:= TRUE;
				SC_OvlZdvihu.Step:= 0;
			END_IF

		40:
			SC_OvlZdvihu.StepName:= '40 - Polohovanie';
			SC_OvlZdvihu.IdleTime.PT:= T#500ms;
			SC_OvlZdvihu.AlarmTime.PT:= T#3s;

			ZadanaPoziciaUINT:= LREAL_TO_UINT(P2_Zvaranie.PAR.ServoZdvihu_ZadanaPozicia);
			AktualnaPoziciaUINT:= LREAL_TO_UINT(P2_Zvaranie.STAV.Zdvih_AktualnaPozicia);

			IF NOT SC_OvlZdvihu.Switch1 THEN
				P2_Zvaranie.ServoZdvihuZvarania_M6.CMD.MoveAbsolute:= TRUE;
				SC_OvlZdvihu.Switch1:= TRUE;
			END_IF

			IF (AktualnaPoziciaUINT = ZadanaPoziciaUINT) AND P2_Zvaranie.ServoZdvihuZvarania_M6.STATUS.MoveAbsolute_DONE THEN
				P2_Zvaranie.STAV.ServoZdvihu_PoziciaDosiahnuta:= TRUE;
				SC_OvlZdvihu.ResetStep:= TRUE;
				SC_OvlZdvihu.Step:= 0;
			END_IF

		50:
			SC_OvlZdvihu.StepName:= '50 - Zvaranie';
			SC_OvlZdvihu.IdleTime.PT:= P2_RemPremenne.P2_Zvaranie_CasZvarania;
			SC_OvlZdvihu.AlarmTime.PT:= T#3s;

            P2_Zvaranie.ServoZdvihuZvarania_M6.PAR.Torque:= P2_RemPremenne.P2_Zvaranie_MomentZvarania;
            P2_Zvaranie.ServoZdvihuZvarania_M6.PAR.TorqueAcceleration:= 50;
            P2_Zvaranie.ServoZdvihuZvarania_M6.PAR.TorqueVelocity:= P2_RemPremenne.P2_Zvaranie_RychlostZvarania;
            P2_Zvaranie.ServoZdvihuZvarania_M6.PAR.TorqueRamp;

			SC_OvlZdvihu.IdleTime.IN:= MomentDosiahnuty;

			IF NOT SC_OvlZdvihu.Switch1 THEN
				P2_Zvaranie.ServoZdvihuZvarania_M6.CMD.MoveTorque:= TRUE;
				SC_OvlZdvihu.Switch1:= TRUE;
			END_IF

			IF P2_Zvaranie.ServoZdvihuZvarania_M6.STATUS.ActualTorque >= P2_Zvaranie.ServoZdvihuZvarania_M6.PAR.Torque THEN
				MomentDosiahnuty:= TRUE;
			END_IF

			IF SC_OvlZdvihu.IdleTime.Q THEN
				P2_Zvaranie.STAV.ServoZdvihu_PoziciaDosiahnuta:= TRUE;
				SC_OvlZdvihu.ResetStep:= TRUE;
				SC_OvlZdvihu.Step:= 0;
			END_IF

        60:
            SC_OvlZdvihu.StepName:= '60 - Zatlacanie Coveru 5H';
            SC_OvlZdvihu.IdleTime.PT:= P2_RemPremenne.P2_Zvaranie_CasZatlacania;
            SC_OvlZdvihu.AlarmTime.PT:= T#3s;

            P2_Zvaranie.ServoZdvihuZvarania_M6.PAR.Torque:= P2_RemPremenne.P2_Zvaranie_MomentZatlacania;
            P2_Zvaranie.ServoZdvihuZvarania_M6.PAR.TorqueAcceleration:= 50;
            P2_Zvaranie.ServoZdvihuZvarania_M6.PAR.TorqueVelocity:= P2_RemPremenne.P2_Zvaranie_RychlostZatlacania;
            P2_Zvaranie.ServoZdvihuZvarania_M6.PAR.TorqueRamp;

            SC_OvlZdvihu.IdleTime.IN:= MomentDosiahnuty;

            IF NOT SC_OvlZdvihu.Switch1 THEN
                P2_Zvaranie.ServoZdvihuZvarania_M6.CMD.MoveTorque:= TRUE;
                SC_OvlZdvihu.Switch1:= TRUE;
            END_IF

            IF P2_Zvaranie.ServoZdvihuZvarania_M6.STATUS.ActualTorque >= P2_Zvaranie.ServoZdvihuZvarania_M6.PAR.Torque THEN
                MomentDosiahnuty:= TRUE;
            END_IF

            IF SC_OvlZdvihu.IdleTime.Q THEN
                P2_Zvaranie.STAV.ServoZdvihu_PoziciaDosiahnuta:= TRUE;
                SC_OvlZdvihu.ResetStep:= TRUE;
                SC_OvlZdvihu.Step:= 0;
            END_IF

	END_CASE

END_ACTION
```

#### OvlPojazdu.st
```iecst
ACTION OvlPojazdu:

	//Volanie funkcie SequenceControl//
	SequenceControl(SC:= SC_OvlPojazdu);

	CASE SC_OvlPojazdu.Step OF

		0:
			SC_OvlPojazdu.StepName:= '0 - Nulovanie';
			PresunVPRAVO:= FALSE;
			PresunVLAVO:= FALSE;
			P2_Zvaranie.OUT.PojazdZvarania_VPRAVO_YV45:= FALSE;
			P2_Zvaranie.OUT.PojazdZvarania_VLAVO_YV46:= FALSE;

			IF SC_P2_Zvaranie.Step <> 0 THEN
				SC_OvlPojazdu.ResetStep:= TRUE;
				SC_OvlPojazdu.Step:= 1;
			END_IF

		1:
			SC_OvlPojazdu.StepName:= '1 - Rozhodnutie o cinnosti';
			IF PresunVPRAVO THEN
				SC_OvlPojazdu.Step:= 10;
			ELSIF PresunVLAVO THEN
				SC_OvlPojazdu.Step:= 20;
			END_IF

		10:
			SC_OvlPojazdu.StepName:= '10 - Presunutie zvaracky vpravo';
			SC_OvlPojazdu.IdleTime.PT:= T#3s;
			SC_OvlPojazdu.AlarmTime.PT:= T#3s;

			IF P2_Zvaranie.Automat THEN
				SC_OvlPojazdu.AlarmTime.IN:= TRUE;
			ELSE
				SC_OvlPojazdu.IdleTime.IN:= TRUE;
			END_IF

			IF NOT SC_OvlPojazdu.Switch1 THEN
				P2_Zvaranie.OUT.PojazdZvarania_VPRAVO_YV45:= TRUE;
				SC_OvlPojazdu.Switch1:= TRUE;
			END_IF

			IF P2_Zvaranie.IN.PojazdZvarania_PozVPRAVO_IS10 OR SC_OvlPojazdu.IdleTime.Q THEN
				SC_OvlPojazdu.ResetStep:= TRUE;
				SC_OvlPojazdu.Step:= 0;
			ELSIF SC_OvlPojazdu.AlarmTime.Q THEN
				P2_Alarmy[221]:= TRUE;
			END_IF

		20:
			SC_OvlPojazdu.StepName:= '20 - Presunutie zvaracky vlavo';
			SC_OvlPojazdu.IdleTime.PT:= T#3s;
			SC_OvlPojazdu.AlarmTime.PT:= T#3s;

			IF P2_Zvaranie.Automat THEN
				SC_OvlPojazdu.AlarmTime.IN:= TRUE;
			ELSE
				SC_OvlPojazdu.IdleTime.IN:= TRUE;
			END_IF

			IF NOT SC_OvlPojazdu.Switch1 THEN
				P2_Zvaranie.OUT.PojazdZvarania_VLAVO_YV46:= TRUE;
				SC_OvlPojazdu.Switch1:= TRUE;
			END_IF

			IF P2_Zvaranie.IN.PojazdZvarania_PozVLAVO_IS11 OR SC_OvlPojazdu.IdleTime.Q THEN
				SC_OvlPojazdu.ResetStep:= TRUE;
				SC_OvlPojazdu.Step:= 0;
			ELSIF SC_OvlPojazdu.AlarmTime.Q THEN
				P2_Alarmy[221]:= TRUE;
			END_IF

	END_CASE

END_ACTION
```

### Program Logical/Program/Pracovisko_2/P2_Cistenie (IEC)

#### Main.st - Init, cyclic, exit code
```iecst
PROGRAM _INIT
	(* Insert code here *)

END_PROGRAM

PROGRAM _CYCLIC

	//Volanie funkcie SequenceControl//
	SequenceControl(SC:= SC_P2_Cistenie);

	//Volanie podprogramov//
	OvlDveri;

	//Reset sekcie //
    IF NOT Safety.STAV.P2_ZonaBunky_AKTIVNA THEN
        SC_P2_Cistenie.Step:= 0;
    ELSIF P2_Cistenie.Reset THEN
		SC_P2_Cistenie.Step:= 0;
		P2_Cistenie.Reset:= FALSE;
	END_IF

    CASE SC_P2_Cistenie.Step OF

		0:
			SC_P2_Cistenie.StepName:='0 - Nulovanie';
			SC_OvlDveri.Step:= 0;
			P2_Cistenie.Automat:= FALSE;
			P2_Cistenie.KoniecCyklu:= FALSE;
			P2_Cistenie.Manual:= FALSE;
			P2_Cistenie.STAV.PoINIT:= FALSE;
			P2_Cistenie.OUT.Ionizator_RUN_ZX2:= FALSE;
			P2_Cistenie.OUT.Odsavanie_OfukRUN_YV50:= FALSE;
			P2_Cistenie.OUT.Odsavanie_RUN_YV49:= FALSE;
			P2_Cistenie.OUT.VzduchPreIonizator_RUN_YV51:= FALSE;
			P2_Robot.KOM_OUT.Cistenie_BezpecnaPozicia:= FALSE;
			P2_Robot.KOM_OUT.Cistenie_OdoberPowerCP_4F:= FALSE;
			P2_Robot.KOM_OUT.Cistenie_OdoberPowerCP_5F:= FALSE;
			P2_Robot.KOM_OUT.Cistenie_OdoberPowerCP_5H:= FALSE;
			P2_Robot.KOM_OUT.Cistenie_OtacajPowerCP:= FALSE;
			P2_Robot.KOM_OUT.Cistenie_PolozPowerCP_4F:= FALSE;
			P2_Robot.KOM_OUT.Cistenie_PolozPowerCP_5F:= FALSE;
			P2_Robot.KOM_OUT.Cistenie_PolozPowerCP_5H:= FALSE;

			IF Safety.STAV.P2_ZonaBunky_AKTIVNA AND NOT P2_Pracovisko.STAV.PORUCHA AND P2_Pracovisko.IN.PrivodVzduchu_SnimacTlaku_S3 THEN
				SC_P2_Cistenie.ResetStep:= TRUE;
				SC_P2_Cistenie.Step:= 1;
			END_IF

		1:
			SC_P2_Cistenie.StepName:='1 - Cakam na spustenie vyroby';
			P2_Cistenie.KoniecCyklu:= FALSE;
            IF P2_Cistenie.Automat THEN
				SC_P2_Cistenie.Step:= 2;
			ELSIF P2_Cistenie.Manual THEN
				SC_P2_Cistenie.Step:= 700;
			END_IF

			//********************************************************Inicializácia****************************************************************************//

		2:
			SC_P2_Cistenie.StepName:='2 - Inicializacia - cakam na spustenie inicializacie';
			SC_P2_Cistenie.IdleTime.PT:= T#500ms;
			SC_P2_Cistenie.AlarmTime.PT:= T#5s;
			SC_P2_Cistenie.IdleTime.IN:= TRUE;

			IF SC_P2_Cistenie.IdleTime.Q THEN
				SC_P2_Cistenie.ResetStep:= TRUE;
				SC_P2_Cistenie.Step:= 3;
			END_IF

		3:
			SC_P2_Cistenie.StepName:='2 - Inicializacia - otvorenie dveri';
			SC_P2_Cistenie.IdleTime.PT:= T#500ms;
			SC_P2_Cistenie.AlarmTime.PT:= T#5s;

			IF NOT SC_P2_Cistenie.Switch1 THEN
				Dvere_OTVOR:= TRUE;
				SC_P2_Cistenie.Switch1:= TRUE;
			END_IF

			IF P2_Cistenie.IN.Dvere_OTVORENE_MS7 THEN
				P2_Robot.KOM_OUT.Cistenie_BezpecnaPozicia:= TRUE;
				P2_Cistenie.STAV.PoINIT:= TRUE;
				SC_P2_Cistenie.ResetStep:= TRUE;
				SC_P2_Cistenie.Step:= 100;
			END_IF

			//********************************************************Automatický režim****************************************************************************//

		100:
			SC_P2_Cistenie.StepName:='100 - Automaticky Rezim - cakam na spustenie cistenia';
			SC_P2_Cistenie.IdleTime.PT:= T#200ms;
			SC_P2_Cistenie.AlarmTime.PT:= T#5s;

            IF P2_Cistenie.KoniecCyklu AND NOT P2_StoperZvarania.Automat THEN
                SC_P2_Cistenie.ResetStep:= TRUE;
                SC_P2_Cistenie.Step:= 0;
            ELSIF P2_StoperZvarania.OUT.KOM_Cistenie_START THEN
				SC_P2_Cistenie.ResetStep:= TRUE;
				SC_P2_Cistenie.Step:= 102;
			END_IF

		102:
			SC_P2_Cistenie.StepName:='102 - Automaticky Rezim - vystavenie signalu pre robota odober Power CP z paletky a presun do cistenia';
			SC_P2_Cistenie.IdleTime.PT:= T#200ms;
			SC_P2_Cistenie.AlarmTime.PT:= T#5s;

			IF NOT P2_Robot.KOM_IN.Stav_Cistenie_PowerCP_v_Cisteni AND NOT P2_Cistenie.IN.VakumDosiahnute_S5 THEN
				P2_Robot.KOM_OUT.Cistenie_BezpecnaPozicia:= TRUE;
				IF Linka.PAR.ZvolenyModel = '4F' THEN
					P2_Robot.KOM_OUT.Cistenie_OdoberPowerCP_4F:= TRUE;
					P2_Cistenie.OUT.Odsavanie_RUN_YV49:= TRUE;
					SC_P2_Cistenie.ResetStep:= TRUE;
					SC_P2_Cistenie.Step:= 105;
				ELSIF Linka.PAR.ZvolenyModel = '5F' THEN
					P2_Robot.KOM_OUT.Cistenie_OdoberPowerCP_5F:= TRUE;
					P2_Cistenie.OUT.Odsavanie_RUN_YV49:= TRUE;
					SC_P2_Cistenie.ResetStep:= TRUE;
					SC_P2_Cistenie.Step:= 105;
				ELSIF Linka.PAR.ZvolenyModel = '5H' THEN
					P2_Robot.KOM_OUT.Cistenie_OdoberPowerCP_5H:= TRUE;
					P2_Cistenie.OUT.Odsavanie_RUN_YV49:= TRUE;
					SC_P2_Cistenie.ResetStep:= TRUE;
					SC_P2_Cistenie.Step:= 105;
				END_IF
			END_IF

		105:
			SC_P2_Cistenie.StepName:='105 - Automaticky Rezim - cakam na signal robot odobral Power CP z paletky';
			SC_P2_Cistenie.IdleTime.PT:= T#200ms;
			SC_P2_Cistenie.AlarmTime.PT:= T#5s;

			IF P2_Robot.KOM_IN.Stav_Cistenie_PowerCP_v_Cisteni THEN
				P2_Robot.KOM_OUT.Cistenie_OdoberPowerCP_4F:= FALSE;
				P2_Robot.KOM_OUT.Cistenie_OdoberPowerCP_5F:= FALSE;
				P2_Robot.KOM_OUT.Cistenie_OdoberPowerCP_5H:= FALSE;
				SC_P2_Cistenie.ResetStep:= TRUE;
				SC_P2_Cistenie.Step:= 108;
			END_IF

		108:
			SC_P2_Cistenie.StepName:='108 - Automaticky Rezim - zatvorenie dveri, spustenie ionizatora';
			SC_P2_Cistenie.IdleTime.PT:= T#2s;
			SC_P2_Cistenie.AlarmTime.PT:= T#5s;

			IF NOT SC_P2_Cistenie.Switch1 THEN
				P2_Cistenie.OUT.Ionizator_RUN_ZX2:= TRUE;
				P2_Cistenie.OUT.VzduchPreIonizator_RUN_YV51:= TRUE;
				Dvere_ZATVOR:= TRUE;
				P2_Robot.KOM_OUT.Cistenie_BezpecnaPozicia:= FALSE;
				SC_P2_Cistenie.Switch1:= TRUE;
			END_IF

			IF P2_Cistenie.IN.Dvere_ZATVORENE_MS8 THEN
				P2_Cistenie.OUT.Ionizator_RUN_ZX2:= FALSE;
				P2_Cistenie.OUT.VzduchPreIonizator_RUN_YV51:= FALSE;
				SC_P2_Cistenie.ResetStep:= TRUE;
				SC_P2_Cistenie.Step:= 112;
			END_IF

		112:
			SC_P2_Cistenie.StepName:='112 - Automaticky Rezim - zapnutie ofuku';
			SC_P2_Cistenie.IdleTime.PT:= T#2s;
			SC_P2_Cistenie.AlarmTime.PT:= T#5s;

			IF P2_Cistenie.IN.VakumDosiahnute_S5 THEN
				P2_Cistenie.OUT.Odsavanie_OfukRUN_YV50:= TRUE;
				SC_P2_Cistenie.ResetStep:= TRUE;
				SC_P2_Cistenie.Step:= 115;
			END_IF

		115:
			SC_P2_Cistenie.StepName:='115 - Automaticky Rezim - vystavenie signalu pre robota vykonaj otacanie Power CP v cisteni';
			SC_P2_Cistenie.IdleTime.PT:= T#200ms;
			SC_P2_Cistenie.AlarmTime.PT:= T#5s;

			IF NOT P2_Robot.KOM_IN.Stav_Cistenie_Otacanie_Ukoncene THEN
				P2_Robot.KOM_OUT.Cistenie_OtacajPowerCP:= TRUE;
				SC_P2_Cistenie.ResetStep:= TRUE;
				SC_P2_Cistenie.Step:= 118;
			END_IF

		118:
			SC_P2_Cistenie.StepName:='118 - Automaticky Rezim - cakam na signal robot ukoncil otacanie Power CP';
			SC_P2_Cistenie.IdleTime.PT:= T#200ms;
			SC_P2_Cistenie.AlarmTime.PT:= T#5s;

			IF P2_Robot.KOM_IN.Stav_Cistenie_Otacanie_Ukoncene THEN
				P2_Robot.KOM_OUT.Cistenie_OtacajPowerCP:= FALSE;
				SC_P2_Cistenie.ResetStep:= TRUE;
				SC_P2_Cistenie.Step:= 120;
			END_IF

		120:
			SC_P2_Cistenie.StepName:='120 - Automaticky Rezim - otvorenie dveri,vypnutie ofuku a odsavania';
			SC_P2_Cistenie.IdleTime.PT:= T#2s;
			SC_P2_Cistenie.AlarmTime.PT:= T#5s;

			IF NOT SC_P2_Cistenie.Switch1 THEN
				P2_Cistenie.OUT.Odsavanie_OfukRUN_YV50:= FALSE;
				P2_Cistenie.OUT.Odsavanie_RUN_YV49:= FALSE;
				Dvere_OTVOR:= TRUE;
				SC_P2_Cistenie.Switch1:= TRUE;
			END_IF

			IF P2_Cistenie.IN.Dvere_OTVORENE_MS7 THEN
				P2_Robot.KOM_OUT.Cistenie_BezpecnaPozicia:= TRUE;
				SC_P2_Cistenie.ResetStep:= TRUE;
				SC_P2_Cistenie.Step:= 122;
			END_IF

		122:
			SC_P2_Cistenie.StepName:='122 - Automaticky Rezim - vystavenie signalu pre robota poloz Power CP na paletku po cisteni';
			SC_P2_Cistenie.IdleTime.PT:= T#200ms;
			SC_P2_Cistenie.AlarmTime.PT:= T#5s;

			IF NOT P2_Robot.KOM_IN.Stav_Cistenie_PowerCP_Polozene THEN
				IF Linka.PAR.ZvolenyModel = '4F' THEN
					P2_Robot.KOM_OUT.Cistenie_PolozPowerCP_4F:= TRUE;
					SC_P2_Cistenie.ResetStep:= TRUE;
					SC_P2_Cistenie.Step:= 125;
				ELSIF Linka.PAR.ZvolenyModel = '5F' THEN
					P2_Robot.KOM_OUT.Cistenie_PolozPowerCP_5F:= TRUE;
					SC_P2_Cistenie.ResetStep:= TRUE;
					SC_P2_Cistenie.Step:= 125;
				ELSIF Linka.PAR.ZvolenyModel = '5H' THEN
					P2_Robot.KOM_OUT.Cistenie_PolozPowerCP_5H:= TRUE;
					SC_P2_Cistenie.ResetStep:= TRUE;
					SC_P2_Cistenie.Step:= 125;
				END_IF
			END_IF

		125:
			SC_P2_Cistenie.StepName:='125 - Automaticky Rezim - cakam na signal robot polozil Power CP na paletku';
			SC_P2_Cistenie.IdleTime.PT:= T#200ms;
			SC_P2_Cistenie.AlarmTime.PT:= T#5s;

			IF P2_Robot.KOM_IN.Stav_Cistenie_PowerCP_Polozene THEN
				P2_Robot.KOM_OUT.Cistenie_PolozPowerCP_4F:= FALSE;
				P2_Robot.KOM_OUT.Cistenie_PolozPowerCP_5F:= FALSE;
				P2_Robot.KOM_OUT.Cistenie_PolozPowerCP_5H:= FALSE;
				SC_P2_Cistenie.ResetStep:= TRUE;
				SC_P2_Cistenie.Step:= 128;
			END_IF

		128:
			SC_P2_Cistenie.StepName:='122 - Automaticky Rezim - vystavenie signalu ukoncenie cistenia';
			SC_P2_Cistenie.IdleTime.PT:= T#200ms;
			SC_P2_Cistenie.AlarmTime.PT:= T#5s;

			IF NOT SC_P2_Cistenie.Switch1 THEN
				P2_Cistenie.OUT.KOM_CistenieUkoncene:= TRUE;
				SC_P2_Cistenie.Switch1:= TRUE;
			END_IF

			IF NOT P2_StoperZvarania.OUT.KOM_Cistenie_START THEN
				SC_P2_Cistenie.ResetStep:= TRUE;
				SC_P2_Cistenie.Step:= 100;
			END_IF

	END_CASE

END_PROGRAM

PROGRAM _EXIT
	(* Insert code here *)

END_PROGRAM
```

#### Variables.var - Local variables
```iecst
VAR
	SC_OvlDveri : SequenceControlTyp;
	Dvere_OTVOR : BOOL;
	Dvere_ZATVOR : BOOL;
END_VAR
```

#### OvlDveri.st
```iecst
ACTION OvlDveri:

	//Volanie funkcie SequenceControl//
	SequenceControl(SC:= SC_OvlDveri);

	CASE SC_OvlDveri.Step OF

		0:
			SC_OvlDveri.StepName:= '0 - Nulovanie';
			Dvere_OTVOR:= FALSE;
			Dvere_ZATVOR:= FALSE;
			P2_Cistenie.OUT.Dvere_OTVOR_YV47:= FALSE;
			P2_Cistenie.OUT.Dvere_ZATVOR_YV48:= FALSE;

			IF SC_P2_Cistenie.Step <> 0 THEN
				SC_OvlDveri.ResetStep:= TRUE;
				SC_OvlDveri.Step:= 1;
			END_IF

		1:
			SC_OvlDveri.StepName:= '1 - Rozhodnutie o cinnosti';
			IF Dvere_OTVOR THEN
				SC_OvlDveri.Step:= 10;
			ELSIF Dvere_ZATVOR THEN
				SC_OvlDveri.Step:= 20;
			END_IF

		10:
			SC_OvlDveri.StepName:= '10 - Otvorenie dveri';
			SC_OvlDveri.IdleTime.PT:= T#3s;
			SC_OvlDveri.AlarmTime.PT:= T#3s;

			IF P2_Cistenie.Automat THEN
				SC_OvlDveri.AlarmTime.IN:= TRUE;
			ELSE
				SC_OvlDveri.IdleTime.IN:= TRUE;
			END_IF

			IF NOT SC_OvlDveri.Switch1 THEN
				P2_Cistenie.OUT.Dvere_OTVOR_YV47:= TRUE;
				SC_OvlDveri.Switch1:= TRUE;
			END_IF

			IF P2_Cistenie.IN.Dvere_OTVORENE_MS7 OR SC_OvlDveri.IdleTime.Q THEN
				SC_OvlDveri.ResetStep:= TRUE;
				SC_OvlDveri.Step:= 0;
			ELSIF SC_OvlDveri.AlarmTime.Q THEN
				P2_Alarmy[224]:= TRUE;
			END_IF

		20:
			SC_OvlDveri.StepName:= '20 - Zatvorenie dveri';
			SC_OvlDveri.IdleTime.PT:= T#3s;
			SC_OvlDveri.AlarmTime.PT:= T#3s;

			IF P2_Cistenie.Automat THEN
				SC_OvlDveri.AlarmTime.IN:= TRUE;
			ELSE
				SC_OvlDveri.IdleTime.IN:= TRUE;
			END_IF

			IF NOT SC_OvlDveri.Switch1 THEN
				P2_Cistenie.OUT.Dvere_ZATVOR_YV48:= TRUE;
				SC_OvlDveri.Switch1:= TRUE;
			END_IF

			IF P2_Cistenie.IN.Dvere_ZATVORENE_MS8 OR SC_OvlDveri.IdleTime.Q THEN
				SC_OvlDveri.ResetStep:= TRUE;
				SC_OvlDveri.Step:= 0;
			ELSIF SC_OvlDveri.AlarmTime.Q THEN
				P2_Alarmy[223]:= TRUE;
			END_IF

	END_CASE

END_ACTION
```

### Program Logical/Program/Pracovisko_2/P2_OvladanieVizu (IEC)

#### Main.st - Init, cyclic, exit code
```iecst
PROGRAM _INIT

	P2_Vizu.GoPage:= 'PageBootP2';

END_PROGRAM

PROGRAM _CYCLIC

	//************************************Filter alarmov**************************************************************//
	FilterVizu_P2:= '[{"logicalOperator":"and","value":200,"conditionType":">=","columnType":"cod","useAlarmState":false,"alarmState":0},{"value":299,"conditionType":"<=","columnType":"cod","useAlarmState":false,"alarmState":0}]';

	//***********************************Zobrazenie warningov pracoviska****************************************************//
	//0 - Pracovisko je vypnuté.
	//1 - Prebieha inicializácia pracoviska.
	//2 - Na pracovisku prebieha výroba.
	//3 - Prebieha ukončenie pracovného cyklu pracoviska.
	//4 - Prebieha režim vyprázdnenia linky.
	//5 - Robot nie je prepnuty do automatického režimu !!!
	//6 - Doplň zásobník matíc M4 !!!
	//7 - Doplň zásobník skrutiek M4 !!!
	//8 - Doplň zásobník skrutiek M5 !!!
	//9 - Doplň zásobník skrutiek M6 !!!

	IF NOT P2_Robot.KOM_IN.Stav_RezimAUTOMAT THEN
		P2_Vizu.Warnings_Index:= 5;
	ELSIF P2_SkrutkovacMatic.STAV.Zasobnik_Matic_M4_Prazdny THEN
		P2_Vizu.Warnings_Index:= 6;
	ELSIF P2_Srobovanie.STAV.Zasobnik_M4_Prazdny THEN
		P2_Vizu.Warnings_Index:= 7;
	ELSIF P2_Srobovanie.STAV.Zasobnik_M5_Prazdny THEN
		P2_Vizu.Warnings_Index:= 8;
	ELSIF P2_Srobovanie.STAV.Zasobnik_M6_Prazdny THEN
        P2_Vizu.Warnings_Index:= 9;
    ELSIF Linka.TestovaciKus THEN
        P2_Vizu.Warnings_Index:= 11;
	ELSIF Linka.VyprazdnenieLinky THEN
		P2_Vizu.Warnings_Index:= 4;
	ELSIF P2_Pracovisko.STAV.Automat AND NOT P2_Pracovisko.STAV.PoINIT AND NOT P2_Pracovisko.STAV.UkoncenieCyklu_BUSY THEN
		P2_Vizu.Warnings_Index:= 1;
	ELSIF P2_Pracovisko.STAV.PoINIT AND NOT P2_Pracovisko.STAV.UkoncenieCyklu_BUSY THEN
		P2_Vizu.Warnings_Index:= 2;
	ELSIF P2_Pracovisko.STAV.UkoncenieCyklu_BUSY THEN
		P2_Vizu.Warnings_Index:= 3;
	ELSIF NOT P2_Pracovisko.STAV.Automat THEN
		P2_Vizu.Warnings_Index:= 0;
	END_IF

	//************************Prepínanie farby textového pola warning zariadenia***********************************//
	IF P2_Vizu.Warnings_Index = 0 THEN
		P2_Vizu.Warnings_Farba:= "TextOutput_Green";
	ELSIF P2_Vizu.Warnings_Index = 1 THEN
		P2_Vizu.Warnings_Farba:= "TextOutput_Green";
	ELSIF P2_Vizu.Warnings_Index = 2 THEN
		P2_Vizu.Warnings_Farba:= "TextOutput_Green";
	ELSIF P2_Vizu.Warnings_Index = 3 THEN
		P2_Vizu.Warnings_Farba:= "TextOutput_Green";
	ELSIF P2_Vizu.Warnings_Index = 4 THEN
        P2_Vizu.Warnings_Farba:= "TextOutput_Green";
    ELSIF P2_Vizu.Warnings_Index = 11 THEN
        P2_Vizu.Warnings_Farba:= "TextOutput_Green";
	ELSE
		IF Blikac1s THEN
			P2_Vizu.Warnings_Farba:= "TextOutput_Red";
		ELSE
			P2_Vizu.Warnings_Farba:= "TextOutput_Grey";
		END_IF
	END_IF

    //***********************Prepnutie na obrazovku Automat z ručného režimu******************//
    IF P2_Pracovisko.STAV.Manual AND NOT Safety.STAV.P2_ZamkyBunky_AKTIVNE THEN
        P2_Pracovisko.Reset:= TRUE;
        P2_Vizu.GoPage:= 'PageBootP2';
    END_IF

	//***********************Prepnutie bootovacej obrazovky********************************//
	IF NOT Safety.STAV.SafetyPLC_Nabehlo THEN
        P2_Vizu.GoPage:= 'PageBootP2';
    ELSIF CasPrepnutiaObrazovky.Q THEN
        P2_Vizu.GoPage:= 'PageBootP2';
	ELSIF P2_Vizu.ActualPage = 'PageBootP2' AND Safety.STAV.SafetyPLC_Nabehlo THEN
		P2_Vizu.GoPage:= 'PageAutomatP2';
	END_IF

    CasPrepnutiaObrazovky.IN:= P2_Vizu.ActualPage = 'PageBootP2' AND P2_Vizu.GoPage = 'PageAutomatP2';
    CasPrepnutiaObrazovky.PT:= T#5s;
    CasPrepnutiaObrazovky();

	//*************************************Zamknutie tlačítok***************************************************************//
	//Tlačítko Štat Automat//
	IF P2_Pracovisko.STAV.UkoncenieCyklu_BUSY THEN
        P2_Vizu.TL_StartAutomat_ENABLE:= FALSE;
    ELSIF P2_Pracovisko.STAV.PORUCHA THEN
        P2_Vizu.TL_StartAutomat_ENABLE:= FALSE;
    ELSIF NOT P2_Robot.KOM_IN.Stav_RezimAUTOMAT THEN
		P2_Vizu.TL_StartAutomat_ENABLE:= FALSE;
	ELSIF NOT Safety.STAV.P2_ZonaBunky_AKTIVNA THEN
		P2_Vizu.TL_StartAutomat_ENABLE:= FALSE;
    ELSE
        P2_Vizu.TL_StartAutomat_ENABLE:= TRUE;
    END_IF

	//Tlačítko Ukončenie Cyklu//
	IF P2_Pracovisko.STAV.PoINIT THEN
		P2_Vizu.TL_KoniecCyklu_ENABLE:= TRUE;
	ELSE
		P2_Vizu.TL_KoniecCyklu_ENABLE:= FALSE;
	END_IF

    //Tlačítko STOP//
    IF P2_Pracovisko.STAV.PoINIT THEN
        P2_Vizu.TL_STOP_ENABLE:= FALSE;
    ELSE
        P2_Vizu.TL_STOP_ENABLE:= TRUE;
    END_IF

	//Tlačítko Režim Automat//
	P2_Vizu.TL_RezimAutomat_ENABLE:= TRUE;

    //Tlačítko Režim Manual//
	IF P2_Pracovisko.STAV.Automat THEN
		P2_Vizu.TL_RezimManual_ENABLE:= FALSE;
	ELSIF NOT P2_Pracovisko.STAV.Manual AND NOT P2_Pracovisko.STAV.READY THEN
        P2_Vizu.TL_RezimManual_ENABLE:= FALSE;
    ELSIF NOT Safety.STAV.P2_ZamkyBunky_AKTIVNE THEN
        P2_Vizu.TL_RezimManual_ENABLE:= FALSE;
	ELSE
		P2_Vizu.TL_RezimManual_ENABLE:= TRUE;
	END_IF

	//Tlačítka ovládania zámkov//
	IF NOT P2_Pracovisko.STAV.Automat THEN
		P2_Vizu.TL_OvladaniaZamkov_ENABLE:= TRUE;
	ELSE
		P2_Vizu.TL_OvladaniaZamkov_ENABLE:= FALSE;
	END_IF

	//Tlačítko ovládania zdvihu zakladača tesnenia//
	IF NOT P2_ZakladacTesnenia.STAV.ServoZdvihu_HomingOK THEN
        P2_Vizu.ZaklTesnenia_OvlZdvihu_ENABLE:= FALSE;
    ELSIF NOT Safety.STAV.P2_ZaklTesnenia_Pojazd_ZASUNUTY THEN
        P2_Vizu.ZaklTesnenia_OvlZdvihu_ENABLE:= FALSE;
    ELSIF NOT Safety.STAV.P2_ZaklTesnenia_Bariera_AKTIVNA THEN
        P2_Vizu.ZaklTesnenia_OvlZdvihu_ENABLE:= FALSE;
	ELSE
		P2_Vizu.ZaklTesnenia_OvlZdvihu_ENABLE:= TRUE;
	END_IF

	//Tlačítko ovládania zostupu zakladača tesnenia//
	IF NOT P2_ZakladacTesnenia.STAV.ServoZdvihu_HomingOK THEN
		P2_Vizu.ZaklTesnenia_OvlZostupu_ENABLE:= FALSE;
	ELSIF NOT Safety.STAV.P2_ZaklTesnenia_Pojazd_ZASUNUTY THEN
        P2_Vizu.ZaklTesnenia_OvlZostupu_ENABLE:= FALSE;
    ELSIF NOT Safety.STAV.P2_ZaklTesnenia_Bariera_AKTIVNA THEN
        P2_Vizu.ZaklTesnenia_OvlZostupu_ENABLE:= FALSE;
	ELSE
		P2_Vizu.ZaklTesnenia_OvlZostupu_ENABLE:= TRUE;
	END_IF

	//Tlačítka ovládania pojazdu zakladača tesnenia//
	IF NOT P2_ZakladacTesnenia.STAV.ServoPojazdu_HomingOK THEN
		P2_Vizu.ZaklTesnenia_OvlPojazdu_ENABLE:= FALSE;
	ELSIF P2_ZakladacTesnenia.STAV.Zdvih_AktualnaPozicia > 5 THEN
        P2_Vizu.ZaklTesnenia_OvlPojazdu_ENABLE:= FALSE;
    ELSE
		P2_Vizu.ZaklTesnenia_OvlPojazdu_ENABLE:= TRUE;
	END_IF

	//Tlačítka ovládanie osy X manipulátora šróbovačiek//
	IF NOT P2_Srobovanie.STAV.OsX_HomingOK THEN
        P2_Vizu.Srobovanie_OvlManipOsX_ENABLE:= FALSE;
    ELSIF NOT P2_Srobovacky_VychodziaPozicia THEN
        P2_Vizu.Srobovanie_OvlManipOsX_ENABLE:= FALSE;
    ELSIF P2_Srobovanie.RR_PolohujNaPoziciuSkrutky_4F THEN
        P2_Vizu.Srobovanie_OvlManipOsX_ENABLE:= FALSE;
    ELSIF P2_Srobovanie.RR_PolohujNaPoziciuSkrutky_5F THEN
        P2_Vizu.Srobovanie_OvlManipOsX_ENABLE:= FALSE;
    ELSIF P2_Srobovanie.RR_PolohujNaPoziciuSkrutky_5H THEN
        P2_Vizu.Srobovanie_OvlManipOsX_ENABLE:= FALSE;
    ELSIF P2_Srobovanie.STAV.Cistenie_M4_BUSY THEN
        P2_Vizu.Srobovanie_OvlManipOsX_ENABLE:= FALSE;
    ELSIF P2_Srobovanie.STAV.Cistenie_M5_BUSY THEN
        P2_Vizu.Srobovanie_OvlManipOsX_ENABLE:= FALSE;
    ELSIF P2_Srobovanie.STAV.Cistenie_M6_BUSY THEN
        P2_Vizu.Srobovanie_OvlManipOsX_ENABLE:= FALSE;
	ELSE
		P2_Vizu.Srobovanie_OvlManipOsX_ENABLE:= TRUE;
	END_IF

	//Tlačítka ovládania osy Y manipulatora šróbovačiek//
	IF NOT P2_Srobovanie.STAV.OsY_HomingOK THEN
        P2_Vizu.Srobovanie_OvlManipOsY_ENABLE:= FALSE;
    ELSIF NOT P2_Srobovacky_VychodziaPozicia THEN
        P2_Vizu.Srobovanie_OvlManipOsY_ENABLE:= FALSE;
    ELSIF P2_Srobovanie.RR_PolohujNaPoziciuSkrutky_4F THEN
        P2_Vizu.Srobovanie_OvlManipOsY_ENABLE:= FALSE;
    ELSIF P2_Srobovanie.RR_PolohujNaPoziciuSkrutky_5F THEN
        P2_Vizu.Srobovanie_OvlManipOsY_ENABLE:= FALSE;
    ELSIF P2_Srobovanie.RR_PolohujNaPoziciuSkrutky_5H THEN
        P2_Vizu.Srobovanie_OvlManipOsY_ENABLE:= FALSE;
    ELSIF P2_Srobovanie.STAV.Cistenie_M4_BUSY THEN
        P2_Vizu.Srobovanie_OvlManipOsY_ENABLE:= FALSE;
    ELSIF P2_Srobovanie.STAV.Cistenie_M5_BUSY THEN
        P2_Vizu.Srobovanie_OvlManipOsY_ENABLE:= FALSE;
    ELSIF P2_Srobovanie.STAV.Cistenie_M6_BUSY THEN
        P2_Vizu.Srobovanie_OvlManipOsY_ENABLE:= FALSE;
	ELSE
		P2_Vizu.Srobovanie_OvlManipOsY_ENABLE:= TRUE;
	END_IF

	//Tlačítka ovládania zdvihu zvárania//
	IF NOT P2_Zvaranie.STAV.ServoZdvihu_HomingOK THEN
        P2_Vizu.Zvaranie_OvlZdvihu_ENABLE:= FALSE;
    ELSE
		P2_Vizu.Zvaranie_OvlZdvihu_ENABLE:= TRUE;
	END_IF

    //Tlačítka spustenie čistenie skrutkovačiek v ručnom režime//
    IF NOT P2_Srobovacky_VychodziaPozicia THEN
        P2_Vizu.RR_CistenieSkrutkovaciek_ENABLE:= FALSE;
    ELSIF P2_Srobovanie.STAV.Cistenie_M4_BUSY THEN
        P2_Vizu.RR_CistenieSkrutkovaciek_ENABLE:= FALSE;
    ELSIF P2_Srobovanie.STAV.Cistenie_M5_BUSY THEN
        P2_Vizu.RR_CistenieSkrutkovaciek_ENABLE:= FALSE;
    ELSIF P2_Srobovanie.STAV.Cistenie_M6_BUSY THEN
        P2_Vizu.RR_CistenieSkrutkovaciek_ENABLE:= FALSE;
    ELSIF NOT P2_Srobovanie.STAV.OsX_HomingOK THEN
        P2_Vizu.RR_CistenieSkrutkovaciek_ENABLE:= FALSE;
    ELSIF NOT P2_Srobovanie.STAV.OsY_HomingOK THEN
        P2_Vizu.RR_CistenieSkrutkovaciek_ENABLE:= FALSE;
    ELSIF P2_UrovenPrihlasenehoUzivatela < 20 THEN
        P2_Vizu.RR_CistenieSkrutkovaciek_ENABLE:= FALSE;
    ELSIF P2_Srobovanie.RR_PolohujNaPoziciuSkrutky_4F THEN
        P2_Vizu.RR_CistenieSkrutkovaciek_ENABLE:= FALSE;
    ELSIF P2_Srobovanie.RR_PolohujNaPoziciuSkrutky_5F THEN
        P2_Vizu.RR_CistenieSkrutkovaciek_ENABLE:= FALSE;
    ELSIF P2_Srobovanie.RR_PolohujNaPoziciuSkrutky_5H THEN
        P2_Vizu.RR_CistenieSkrutkovaciek_ENABLE:= FALSE;
    ELSE
        P2_Vizu.RR_CistenieSkrutkovaciek_ENABLE:= TRUE;
    END_IF

    //Zamknutie tlačítok test pozicii skrutkovačiek//
    IF NOT P2_Srobovanie.STAV.OsX_HomingOK THEN
        P2_Vizu.RR_PozicieSkrutiek_ENABLE:= FALSE;
    ELSIF NOT P2_Srobovanie.STAV.OsY_HomingOK THEN
        P2_Vizu.RR_PozicieSkrutiek_ENABLE:= FALSE;
    ELSIF NOT P2_Srobovacky_VychodziaPozicia THEN
        P2_Vizu.RR_PozicieSkrutiek_ENABLE:= FALSE;
    ELSIF P2_Srobovanie.STAV.Cistenie_M4_BUSY THEN
        P2_Vizu.RR_PozicieSkrutiek_ENABLE:= FALSE;
    ELSIF P2_Srobovanie.STAV.Cistenie_M5_BUSY THEN
        P2_Vizu.RR_PozicieSkrutiek_ENABLE:= FALSE;
    ELSIF P2_Srobovanie.STAV.Cistenie_M6_BUSY THEN
        P2_Vizu.RR_PozicieSkrutiek_ENABLE:= FALSE;
    ELSIF P2_UrovenPrihlasenehoUzivatela < 100 THEN
        P2_Vizu.RR_PozicieSkrutiek_ENABLE:= FALSE;
    ELSIF P2_Srobovanie.RR_PolohujNaPoziciuSkrutky_4F THEN
        P2_Vizu.RR_PozicieSkrutiek_ENABLE:= FALSE;
    ELSIF P2_Srobovanie.RR_PolohujNaPoziciuSkrutky_5F THEN
        P2_Vizu.RR_PozicieSkrutiek_ENABLE:= FALSE;
    ELSIF P2_Srobovanie.RR_PolohujNaPoziciuSkrutky_5H THEN
        P2_Vizu.RR_PozicieSkrutiek_ENABLE:= FALSE;
    ELSE
        P2_Vizu.RR_PozicieSkrutiek_ENABLE:= TRUE;
    END_IF

	//**************************Zamknutie editácie parametrov*********************************//
    IF P2_UrovenPrihlasenehoUzivatela >= 20 THEN
        P2_Vizu.EditaciaParametrov_ENABLE:= TRUE;
    ELSE
        P2_Vizu.EditaciaParametrov_ENABLE:= FALSE;
    END_IF

	//***************************************Zmena farieb tlačítok pre ovládanie zámkou********************************//
	//Predné dvere pravá strana//
	IF Safety.OUT.P2_ZamkniZamok_PredneDverePS AND Safety.IN.P2_PredneDverePS_PritomPetlice THEN
		P2_Vizu.TL_PrednyZamokPS_Farba:= "Button_Green";
	ELSIF Safety.IN.P2_PredneDverePS_PritomPetlice THEN
		IF Blikac1s THEN
			P2_Vizu.TL_PrednyZamokPS_Farba:= "Button_Blue";
		ELSE
			P2_Vizu.TL_PrednyZamokPS_Farba:= "Operate";
		END_IF
	ELSE
		P2_Vizu.TL_PrednyZamokPS_Farba:= "Button_Red";
	END_IF

	//Predné dvere lavá strana//
	IF Safety.OUT.P2_ZamkniZamok_PredneDvereLS AND Safety.IN.P2_PredneDvereLS_PritomPetlice THEN
		P2_Vizu.TL_PrednyZamokLS_Farba:= "Button_Green";
	ELSIF Safety.IN.P2_PredneDvereLS_PritomPetlice THEN
		IF Blikac1s THEN
			P2_Vizu.TL_PrednyZamokLS_Farba:= "Button_Blue";
		ELSE
			P2_Vizu.TL_PrednyZamokLS_Farba:= "Operate";
		END_IF
	ELSE
		P2_Vizu.TL_PrednyZamokLS_Farba:= "Button_Red";
	END_IF

	//Zadné dvere pravá strana//
	IF Safety.OUT.P2_ZamkniZamok_ZadneDverePS AND Safety.IN.P2_ZadneDverePS_PritomPetlice THEN
		P2_Vizu.TL_ZadnyZamokPS_Farba:= "Button_Green";
	ELSIF Safety.IN.P2_ZadneDverePS_PritomPetlice THEN
		IF Blikac1s THEN
			P2_Vizu.TL_ZadnyZamokPS_Farba:= "Button_Blue";
		ELSE
			P2_Vizu.TL_ZadnyZamokPS_Farba:= "Operate";
		END_IF
	ELSE
		P2_Vizu.TL_ZadnyZamokPS_Farba:= "Button_Red";
	END_IF

	//Zadné dvere lavá strana//
	IF Safety.OUT.P2_ZamkniZamok_ZadneDvereLS AND Safety.IN.P2_ZadneDvereLS_PritomPetlice THEN
		P2_Vizu.TL_ZadnyZamokLS_Farba:= "Button_Green";
	ELSIF Safety.IN.P2_ZadneDvereLS_PritomPetlice THEN
		IF Blikac1s THEN
			P2_Vizu.TL_ZadnyZamokLS_Farba:= "Button_Blue";
		ELSE
			P2_Vizu.TL_ZadnyZamokLS_Farba:= "Operate";
		END_IF
	ELSE
		P2_Vizu.TL_ZadnyZamokLS_Farba:= "Button_Red";
	END_IF

	//***********************************Prepínanie stavov pracovísk*******************************************************************//
	//Dopravníky//
	IF NOT P2_Dopravniky.IN.HornyDoprav_READY OR NOT P2_Dopravniky.IN.SpodnyDoprav_READY THEN
		P2_Vizu.IndexStavu_Dopravnik:= 3;
	ELSIF P2_Dopravniky.Automat AND NOT P2_Dopravniky.STAV.PoINIT THEN
		P2_Vizu.IndexStavu_Dopravnik:= 1;
	ELSIF P2_Dopravniky.Automat AND P2_Dopravniky.STAV.PoINIT THEN
		P2_Vizu.IndexStavu_Dopravnik:= 2;
	ELSE
		P2_Vizu.IndexStavu_Dopravnik:= 0;
	END_IF

	//Stoper zakladania tesnenia//
	IF P2_PoruchaST1 THEN
		P2_Vizu.IndexStavu_StoperZakladacaTesn:= 3;
	ELSIF P2_StoperZaklTesnenia.Automat AND NOT P2_StoperZaklTesnenia.STAV.PoINIT THEN
		P2_Vizu.IndexStavu_StoperZakladacaTesn:= 1;
	ELSIF P2_StoperZaklTesnenia.Automat AND P2_StoperZaklTesnenia.STAV.PoINIT THEN
		P2_Vizu.IndexStavu_StoperZakladacaTesn:= 2;
	ELSE
		P2_Vizu.IndexStavu_StoperZakladacaTesn:= 0;
	END_IF

	//Zakladač tesnenia//
	IF P2_PoruchaST1 THEN
		P2_Vizu.IndexStavu_ZakladacaTesnenia:= 3;
	ELSIF P2_ZakladacTesnenia.Automat AND NOT P2_ZakladacTesnenia.STAV.PoINIT THEN
		P2_Vizu.IndexStavu_ZakladacaTesnenia:= 1;
	ELSIF P2_ZakladacTesnenia.Automat AND P2_ZakladacTesnenia.STAV.PoINIT THEN
		P2_Vizu.IndexStavu_ZakladacaTesnenia:= 2;
	ELSE
		P2_Vizu.IndexStavu_ZakladacaTesnenia:= 0;
	END_IF

	//Stoper maticovačky//
	IF P2_PoruchaST2 THEN
		P2_Vizu.IndexStavu_StoperMaticovacky:= 3;
	ELSIF P2_StoperMaticovacky.Automat AND NOT P2_StoperMaticovacky.STAV.PoINIT THEN
		P2_Vizu.IndexStavu_StoperMaticovacky:= 1;
	ELSIF P2_StoperMaticovacky.Automat AND P2_StoperMaticovacky.STAV.PoINIT THEN
		P2_Vizu.IndexStavu_StoperMaticovacky:= 2;
	ELSE
		P2_Vizu.IndexStavu_StoperMaticovacky:= 0;
	END_IF

	//Stoper šrobovania//
	IF P2_PoruchaST3 THEN
		P2_Vizu.IndexStavu_StoperSrobovania:= 3;
	ELSIF P2_StoperSrobovania.Automat AND NOT P2_StoperSrobovania.STAV.PoINIT THEN
		P2_Vizu.IndexStavu_StoperSrobovania:= 1;
	ELSIF P2_StoperSrobovania.Automat AND P2_StoperSrobovania.STAV.PoINIT THEN
		P2_Vizu.IndexStavu_StoperSrobovania:= 2;
	ELSE
		P2_Vizu.IndexStavu_StoperSrobovania:= 0;
	END_IF

	//Šrobovanie//
	IF P2_PoruchaST3 THEN
		P2_Vizu.IndexStavu_Srobovania:= 3;
	ELSIF P2_Srobovanie.Automat AND NOT P2_Srobovanie.STAV.PoINIT THEN
		P2_Vizu.IndexStavu_Srobovania:= 1;
	ELSIF P2_Srobovanie.Automat AND P2_Srobovanie.STAV.PoINIT THEN
		P2_Vizu.IndexStavu_Srobovania:= 2;
	ELSE
		P2_Vizu.IndexStavu_Srobovania:= 0;
	END_IF

	//Robot//
	IF P2_Robot.Automat AND NOT P2_Robot.STAV.PoINIT THEN
		P2_Vizu.IndexStavu_Robot:= 1;
	ELSIF P2_Robot.Automat AND P2_Robot.STAV.PoINIT THEN
		P2_Vizu.IndexStavu_Robot:= 2;
	ELSE
		P2_Vizu.IndexStavu_Robot:= 0;
	END_IF

	//Stoper zvárania//
	IF P2_PoruchaST4 THEN
		P2_Vizu.IndexStavu_StoperZvarania:= 3;
	ELSIF P2_StoperZvarania.Automat AND NOT P2_StoperZvarania.STAV.PoINIT THEN
		P2_Vizu.IndexStavu_StoperZvarania:= 1;
	ELSIF P2_StoperZvarania.Automat AND P2_StoperZvarania.STAV.PoINIT THEN
		P2_Vizu.IndexStavu_StoperZvarania:= 2;
	ELSE
		P2_Vizu.IndexStavu_StoperZvarania:= 0;
	END_IF

	//Zváranie//
	IF P2_PoruchaST4 THEN
		P2_Vizu.IndexStavu_Zvaranie:= 3;
	ELSIF P2_Zvaranie.Automat AND NOT P2_Zvaranie.STAV.PoINIT THEN
		P2_Vizu.IndexStavu_Zvaranie:= 1;
	ELSIF P2_Zvaranie.Automat AND P2_Zvaranie.STAV.PoINIT THEN
		P2_Vizu.IndexStavu_Zvaranie:= 2;
	ELSE
		P2_Vizu.IndexStavu_Zvaranie:= 0;
	END_IF

	//Čistenie//
	IF P2_PoruchaST4 THEN
		P2_Vizu.IndexStavu_Cistenie:= 3;
	ELSIF P2_Cistenie.Automat AND NOT P2_Cistenie.STAV.PoINIT THEN
		P2_Vizu.IndexStavu_Cistenie:= 1;
	ELSIF P2_Cistenie.Automat AND P2_Cistenie.STAV.PoINIT THEN
		P2_Vizu.IndexStavu_Cistenie:= 2;
	ELSE
		P2_Vizu.IndexStavu_Cistenie:= 0;
	END_IF

END_PROGRAM

PROGRAM _EXIT
	(* Insert code here *)

END_PROGRAM
```

#### Variables.var - Local variables
```iecst
VAR
	CasPrepnutiaObrazovky : TON;
END_VAR
```

### Program Logical/Program/Pracovisko_2/P2_OvladanieSafety (IEC)

#### Main.st - Init, cyclic, exit code
```iecst
PROGRAM _INIT
	(* Insert code here *)

END_PROGRAM

PROGRAM _CYCLIC

	//******************************************Ovládanie zámkov dverí bunky****************************************//
	//Predné dvere - pravá strana//
	IF EDGEPOS(P2_Vizu.TL_ZamkniPrednyZamokPS) THEN
		IF NOT Safety.OUT.P2_ZamkniZamok_PredneDverePS AND Safety.IN.P2_PredneDverePS_PritomPetlice THEN
			Safety.OUT.P2_ZamkniZamok_PredneDverePS:= TRUE;
		ELSIF Safety.OUT.P2_ZamkniZamok_PredneDverePS THEN
			Safety.OUT.P2_ZamkniZamok_PredneDverePS:= FALSE;
		END_IF
		P2_Vizu.TL_ZamkniPrednyZamokPS:= FALSE;
	END_IF

	//Predné dvere - lavá strana//
	IF EDGEPOS(P2_Vizu.TL_ZamkniPrednyZamokLS) THEN
		IF NOT Safety.OUT.P2_ZamkniZamok_PredneDvereLS AND Safety.IN.P2_PredneDvereLS_PritomPetlice THEN
			Safety.OUT.P2_ZamkniZamok_PredneDvereLS:= TRUE;
		ELSIF Safety.OUT.P2_ZamkniZamok_PredneDvereLS THEN
			Safety.OUT.P2_ZamkniZamok_PredneDvereLS:= FALSE;
		END_IF
		P2_Vizu.TL_ZamkniPrednyZamokLS:= FALSE;
	END_IF

	//Zadné dvere - pravá strana//
	IF EDGEPOS(P2_Vizu.TL_ZamkniZadnyZamokPS) THEN
		IF NOT Safety.OUT.P2_ZamkniZamok_ZadneDverePS AND Safety.IN.P2_ZadneDverePS_PritomPetlice THEN
			Safety.OUT.P2_ZamkniZamok_ZadneDverePS:= TRUE;
		ELSIF Safety.OUT.P2_ZamkniZamok_ZadneDverePS THEN
			Safety.OUT.P2_ZamkniZamok_ZadneDverePS:= FALSE;
		END_IF
		P2_Vizu.TL_ZamkniZadnyZamokPS:= FALSE;
	END_IF

	//Zadné dvere - lavá strana//
	IF EDGEPOS(P2_Vizu.TL_ZamkniZadnyZamokLS) THEN
		IF NOT Safety.OUT.P2_ZamkniZamok_ZadneDvereLS AND Safety.IN.P2_ZadneDvereLS_PritomPetlice THEN
			Safety.OUT.P2_ZamkniZamok_ZadneDvereLS:= TRUE;
		ELSIF Safety.OUT.P2_ZamkniZamok_ZadneDvereLS THEN
			Safety.OUT.P2_ZamkniZamok_ZadneDvereLS:= FALSE;
		END_IF
		P2_Vizu.TL_ZamkniZadnyZamokLS:= FALSE;
	END_IF

	//Reset zóny bunky//
	CasResetZonyBunky.IN:= NOT Safety.STAV.P2_ZonaBunky_AKTIVNA	AND Safety.STAV.ZonaCS_AKTIVNA AND Safety.STAV.P2_ZamkyBunky_AKTIVNE AND (Safety.STAV.P3_VstupBunky_Bariera_AKTIVNA OR Safety.STAV.P3_ZamkyBunky_AKTIVNE);

	IF CasResetZonyBunky.Q THEN
		Safety.IN.P2_ZonaBunky_RESET:= TRUE;
	ELSE
		Safety.IN.P2_ZonaBunky_RESET:= FALSE;
	END_IF

	CasResetZonyBunky.PT:= T#1s;
	CasResetZonyBunky();

	//Reset zóny Zakladaca Tesnenia Pojazd//
	CasResetZonyPojazduZaklTesnenia.IN:= NOT Safety.STAV.P2_ZonaZaklTesnenPojazd_AKTIVNA AND Safety.STAV.ZonaCS_AKTIVNA AND (Safety.STAV.P2_ZaklTesnenia_Bumper_AKTIVNY OR NOT Safety.IN.P2_ZaklTesnenia_Vysuvanie_BUSY);

	IF CasResetZonyPojazduZaklTesnenia.Q THEN
		Safety.IN.P2_ZonaZaklTesneniaPojazd_RESET:= TRUE;
	ELSE
		Safety.IN.P2_ZonaZaklTesneniaPojazd_RESET:= FALSE;
	END_IF

	CasResetZonyPojazduZaklTesnenia.PT:= T#1s;
	CasResetZonyPojazduZaklTesnenia();

	//Reset zóny Zakladaca Tesnenia Zdvih//
	CasResetZonyZdvihuZaklTesnenia.IN:= NOT Safety.STAV.P2_ZonaZaklTesnenZdvih_AKTIVNA AND Safety.STAV.ZonaCS_AKTIVNA AND (Safety.STAV.P2_ZaklTesnenia_Bariera_AKTIVNA OR NOT Safety.IN.P2_ZaklTesnenia_Zdvih_BUSY);

	IF CasResetZonyZdvihuZaklTesnenia.Q THEN
		Safety.IN.P2_ZonaZaklTesneniaZdvih_RESET:= TRUE;
	ELSE
		Safety.IN.P2_ZonaZaklTesneniaZdvih_RESET:= FALSE;
	END_IF

	CasResetZonyZdvihuZaklTesnenia.PT:= T#1s;
	CasResetZonyZdvihuZaklTesnenia();

	//Reset zóny Maticovačky//
	CasResetZonyMaticovacky.IN:= NOT Safety.STAV.P2_ZonaMaticovacky_AKTIVNA AND Safety.STAV.ZonaCS_AKTIVNA AND Safety.STAV.P2_ZamkyBunky_AKTIVNE AND Safety.STAV.P2_VstupBunky_Bariera_AKTIVNA;

	IF CasResetZonyMaticovacky.Q THEN
		Safety.IN.P2_ZonaMaticovacky_RESET:= TRUE;
	ELSE
		Safety.IN.P2_ZonaMaticovacky_RESET:= FALSE;
	END_IF

	CasResetZonyMaticovacky.PT:= T#1s;
	CasResetZonyZdvihuZaklTesnenia();

END_PROGRAM

PROGRAM _EXIT
	(* Insert code here *)

END_PROGRAM
```

#### Variables.var - Local variables
```iecst
VAR
	CasResetZonyBunky : TON;
	CasResetZonyPojazduZaklTesnenia : TON;
	CasResetZonyZdvihuZaklTesnenia : TON;
	CasResetZonyMaticovacky : TON;
END_VAR
```

### Program Logical/Program/Pracovisko_3/P3_Main (IEC)

#### Main.st - Init, cyclic, exit code
```iecst
PROGRAM _INIT
	(* Insert code here *)

END_PROGRAM

PROGRAM _CYCLIC

	//Volanie podprogramu//
    OvlVentilovychTerminalov;
    ProfinetKomunikaciaKAM13;

    //******************************Stav moduly OK**************************************//
    IF P3_Pracovisko.STAV.ModulDI31_OK AND
        P3_Pracovisko.STAV.ModulDI32_OK AND
        P3_Pracovisko.STAV.ModulDI33_OK AND
        P3_Pracovisko.STAV.ModulDI34_OK AND
        P3_Pracovisko.STAV.ModulDM31_OK AND
        P3_Pracovisko.STAV.ModulDS31_OK AND
        P3_Pracovisko.STAV.ModulDS32_OK AND
        P3_Pracovisko.STAV.ModulDS33_OK AND
        P3_Pracovisko.STAV.ModulSI31_OK THEN
        P3_Pracovisko.STAV.Moduly_OK:= TRUE;
    ELSE
        P3_Pracovisko.STAV.Moduly_OK:= FALSE;
    END_IF

    //******************************Stav kamery OK**************************************//
    IF Linka.STAV.WenglorControlUnit_OK THEN
        P3_Pracovisko.STAV.Kamery_OK:= TRUE;
    ELSE
        P3_Pracovisko.STAV.Kamery_OK:= FALSE;
    END_IF

    //******************************Stav skrutkovačky OK*********************************//
    IF P3_Pracovisko.STAV.Skrutkovacka_K40_OK AND
        P3_Pracovisko.STAV.Skrutkovacka_M5_OK THEN
        P3_Pracovisko.STAV.Skrutkovacky_OK:= TRUE;
    ELSE
        P3_Pracovisko.STAV.Skrutkovacky_OK:= FALSE;
    END_IF

    //******************************Stav ventilové terminály OK***************************//
    IF P3_Pracovisko.STAV.VentilovyTerminal_VT6_OK AND
        P3_Pracovisko.STAV.VentilovyTerminal_VT7_OK THEN
        P3_Pracovisko.STAV.VentiloveTerminaly_OK:= TRUE;
    ELSE
        P3_Pracovisko.STAV.VentiloveTerminaly_OK:= FALSE;
    END_IF

    //Ukončenie cyklu//
    IF P3_Pracovisko.KoniecCyklu THEN
        IF P3_Dopravniky.Automat THEN
            P3_Dopravniky.KoniecCyklu:= TRUE;
        END_IF
        IF P3_SpodnyStoper.Automat THEN
            P3_SpodnyStoper.KoniecCyklu:= TRUE;
        END_IF
        IF P3_AkumulacnyStoper.Automat THEN
            P3_AkumulacnyStoper.KoniecCyklu:= TRUE;
        END_IF
        IF P3_LeakageTestA.Automat THEN
            P3_LeakageTestA.KoniecCyklu:= TRUE;
        END_IF
        IF P3_LeakageTestB.Automat THEN
            P3_LeakageTestB.KoniecCyklu:= TRUE;
        END_IF
        IF P3_Srobovanie.Automat THEN
            P3_Srobovanie.KoniecCyklu:= TRUE;
        END_IF
        IF P3_StoperSrobovania.Automat THEN
            P3_StoperSrobovania.KoniecCyklu:= TRUE;
        END_IF
        IF P3_VstupnyStoper.Automat THEN
            P3_VstupnyStoper.KoniecCyklu:= TRUE;
        END_IF
        P3_Pracovisko.KoniecCyklu:= FALSE;
    END_IF

    //Ukončenie cyklu pri poruche//
    IF EDGEPOS(P3_PoruchaST1) THEN
        P3_Pracovisko.KoniecCyklu:= TRUE;
    ELSIF EDGEPOS(P3_PoruchaST2) THEN
        P3_Pracovisko.KoniecCyklu:= TRUE;
    ELSIF EDGEPOS(P3_PoruchaST3) THEN
        P3_Pracovisko.KoniecCyklu:= TRUE;
    END_IF

    //Status prebieha ukončenie cyklu//
    IF P3_Dopravniky.KoniecCyklu OR
        P3_SpodnyStoper.KoniecCyklu OR
        P3_AkumulacnyStoper.KoniecCyklu OR
        P3_LeakageTestA.KoniecCyklu OR
        P3_LeakageTestB.KoniecCyklu OR
        P3_Srobovanie.KoniecCyklu OR
        P3_VstupnyStoper.KoniecCyklu OR
        P3_StoperSrobovania.KoniecCyklu THEN
        P3_Pracovisko.STAV.UkoncenieCyklu_BUSY:= TRUE;
    ELSE
        P3_Pracovisko.STAV.UkoncenieCyklu_BUSY:= FALSE;
    END_IF

    //Resetovanie pracoviska  po stlačení tlačítka Automat//
    IF P34_Vizu.TL_RezimAutomat THEN
        IF P3_Pracovisko.STAV.Manual THEN
            P3_Pracovisko.Reset:= TRUE;
        END_IF
        IF P4_Pracovisko.STAV.Manual THEN
            P4_Pracovisko.Reset:= TRUE;
        END_IF
        P34_Vizu.TL_RezimAutomat:= FALSE;
    END_IF

    //Resetovanie pracoviska//
    IF P3_Pracovisko.Reset THEN
        P3_Dopravniky.Reset:= TRUE;
        P3_SpodnyStoper.Reset:= TRUE;
        P3_AkumulacnyStoper.Reset:= TRUE;
        P3_LeakageTestA.Reset:= TRUE;
        P3_LeakageTestB.Reset:= TRUE;
        P3_Srobovanie.Reset:= TRUE;
        P3_StoperSrobovania.Reset:= TRUE;
        P3_VstupnyStoper.Reset:= TRUE;
        P3_Pracovisko.Reset:= FALSE;
    END_IF

    //Prepnutie pracoviska do manualneho režimu//
    IF P3_Pracovisko.Manual THEN
        P3_Dopravniky.Manual:= TRUE;
        P3_SpodnyStoper.Manual:= TRUE;
        P3_AkumulacnyStoper.Manual:= TRUE;
        P3_LeakageTestA.Manual:= TRUE;
        P3_LeakageTestB.Manual:= TRUE;
        P3_Srobovanie.Manual:= TRUE;
        P3_StoperSrobovania.Manual:= TRUE;
        P3_VstupnyStoper.Manual:= TRUE;
        P3_Pracovisko.Manual:= FALSE;
    END_IF

    //Spustenie pracoviska v automatickom režime//
    IF P3_Pracovisko.Automat THEN
        P3_Dopravniky.Automat:= TRUE;
        P3_SpodnyStoper.Automat:= TRUE;
        P3_AkumulacnyStoper.Automat:= TRUE;
        P3_LeakageTestA.Automat:= TRUE;
        P3_LeakageTestB.Automat:= TRUE;
        P3_Srobovanie.Automat:= TRUE;
        P3_StoperSrobovania.Automat:= TRUE;
        P3_VstupnyStoper.Automat:= TRUE;
        P3_Pracovisko.Automat:= FALSE;
    END_IF

    //***********************************Príznaky pracoviska****************************************//
    //Príznak pracovisko stav AUTOMAT//
    IF P3_Dopravniky.Automat OR
        P3_SpodnyStoper.Automat OR
        P3_AkumulacnyStoper.Automat OR
        P3_LeakageTestA.Automat OR
        P3_LeakageTestB.Automat OR
        P3_Srobovanie.Automat OR
        P3_VstupnyStoper.Automat OR
        P3_StoperSrobovania.Automat THEN
        P3_Pracovisko.STAV.Automat:= TRUE;
    ELSE
        P3_Pracovisko.STAV.Automat:= FALSE;
    END_IF

    //Priznak pracovisko stav MANUAL//
    IF P3_Dopravniky.Manual OR
        P3_SpodnyStoper.Manual OR
        P3_AkumulacnyStoper.Manual OR
        P3_LeakageTestA.Manual OR
        P3_LeakageTestB.Manual OR
        P3_Srobovanie.Manual OR
        P3_VstupnyStoper.Manual OR
        P3_StoperSrobovania.Manual THEN
        P3_Pracovisko.STAV.Manual:= TRUE;
    ELSE
        P3_Pracovisko.STAV.Manual:= FALSE;
    END_IF

    //Príznak pracovisko stav PoINIT//
    IF P3_Dopravniky.STAV.PoINIT AND
        P3_SpodnyStoper.STAV.PoINIT AND
        P3_AkumulacnyStoper.STAV.PoINIT AND
        P3_LeakageTestA.STAV.PoINIT AND
        P3_LeakageTestB.STAV.PoINIT AND
        P3_Srobovanie.STAV.PoINIT AND
        P3_VstupnyStoper.STAV.PoINIT AND
        P3_StoperSrobovania.STAV.PoINIT	THEN
        P3_Pracovisko.STAV.PoINIT:= TRUE;
    ELSE
        P3_Pracovisko.STAV.PoINIT:= FALSE;
    END_IF

    //Príznak pracovisko stav READY//
    IF SC_P3_Dopravniky.Step = 1 AND
        SC_P3_SpodnyStoper.Step = 1 AND
        SC_P3_AkumulacnyStoper.Step = 1 AND
        SC_P3_LeakageTestA.Step = 1 AND
        SC_P3_LeakageTestB.Step = 1 AND
        SC_P3_Srobovanie.Step = 1 AND
        SC_P3_VstupnyStoper.Step = 1 AND
        SC_P3_StoperSrobovania.Step = 1 THEN
        P3_Pracovisko.STAV.READY:= TRUE;
    ELSE
        P3_Pracovisko.STAV.READY:= FALSE;
    END_IF

    //Zapnutie aspoň jedného Leakage Testera//
    IF NOT P3_LeakageTestA.STAV.Tester_ON AND NOT P3_LeakageTestB.STAV.Tester_ON THEN
        P3_LeakageTestB.STAV.Tester_ON:= TRUE;
    END_IF

    //*************************************Zapnutie osvetleniapracoviska****************************************//
    IF NOT Safety.IN.P3_PredneDvereLS_PritomPetlice THEN
        P3_Pracovisko.OUT.OsvetlenieBunky:= TRUE;
    ELSIF NOT Safety.IN.P3_PredneDverePS_PritomPetlice THEN
        P3_Pracovisko.OUT.OsvetlenieBunky:= TRUE;
    ELSIF NOT Safety.IN.P3_ZadneDvere_PritomPetlice THEN
        P3_Pracovisko.OUT.OsvetlenieBunky:= TRUE;
    ELSE
        P3_Pracovisko.OUT.OsvetlenieBunky:= FALSE;
    END_IF

    //****************************************Ovládanie majáka***********************************************//
    //Zelené svetlo//

    IF P3_Pracovisko.STAV.Automat THEN
        P3_Pracovisko.OUT.Majak_ZeleneSvetlo:= TRUE;
    ELSIF P3_Pracovisko.STAV.Manual THEN
        P3_Pracovisko.OUT.Majak_ZeleneSvetlo:= Blikac500ms;
    ELSE
        P3_Pracovisko.OUT.Majak_ZeleneSvetlo:= FALSE;
    END_IF

    //Žlté svetlo//
    IF P3_Pracovisko.STAV.Automat AND NOT P3_Pracovisko.STAV.PoINIT THEN
        P3_Pracovisko.OUT.Majak_ZlteSvetlo:= TRUE;
    ELSIF Linka.PAR.ZvolenyModel = '4F' AND NOT P3_Srobovanie.IN.HVTest_TypKonektoru_4F THEN
        P3_Pracovisko.OUT.Majak_ZlteSvetlo:= Blikac500ms;
    ELSIF Linka.PAR.ZvolenyModel = '5F' AND NOT P3_Srobovanie.IN.HVTest_TypKonektoru_5F_5H THEN
        P3_Pracovisko.OUT.Majak_ZlteSvetlo:= Blikac500ms;
    ELSIF Linka.PAR.ZvolenyModel = '5H' AND NOT P3_Srobovanie.IN.HVTest_TypKonektoru_5F_5H THEN
        P3_Pracovisko.OUT.Majak_ZlteSvetlo:= Blikac500ms;
    ELSIF Linka.PAR.ZvolenyModel = '4F' AND NOT P3_LeakageTestA.IN.Tester_TypKonektoru_4F THEN
        P3_Pracovisko.OUT.Majak_ZlteSvetlo:= Blikac500ms;
    ELSIF Linka.PAR.ZvolenyModel = '5F' AND NOT P3_LeakageTestA.IN.Tester_TypKonektoru_5F_5H THEN
        P3_Pracovisko.OUT.Majak_ZlteSvetlo:= Blikac500ms;
    ELSIF Linka.PAR.ZvolenyModel = '5H' AND NOT P3_LeakageTestA.IN.Tester_TypKonektoru_5F_5H THEN
        P3_Pracovisko.OUT.Majak_ZlteSvetlo:= Blikac500ms;
    ELSIF Linka.PAR.ZvolenyModel = '4F' AND NOT P3_LeakageTestB.IN.Tester_TypKonektoru_4F THEN
        P3_Pracovisko.OUT.Majak_ZlteSvetlo:= Blikac500ms;
    ELSIF Linka.PAR.ZvolenyModel = '5F' AND NOT P3_LeakageTestB.IN.Tester_TypKonektoru_5F_5H THEN
        P3_Pracovisko.OUT.Majak_ZlteSvetlo:= Blikac500ms;
    ELSIF Linka.PAR.ZvolenyModel = '5H' AND NOT P3_LeakageTestB.IN.Tester_TypKonektoru_5F_5H THEN
        P3_Pracovisko.OUT.Majak_ZlteSvetlo:= Blikac500ms;
    ELSIF P3_Srobovanie.STAV.Zasobnik_K40_Prazdny THEN
        P3_Pracovisko.OUT.Majak_ZlteSvetlo:= Blikac500ms;
    ELSIF P3_Srobovanie.STAV.Zasobnik_M5_Prazdny THEN
        P3_Pracovisko.OUT.Majak_ZlteSvetlo:= Blikac500ms;
    ELSE
        P3_Pracovisko.OUT.Majak_ZlteSvetlo:= FALSE;
    END_IF

    //Červené svetlo//
    IF P3_Pracovisko.STAV.PORUCHA THEN
        P3_Pracovisko.OUT.Majak_CerveneSvetlo:= TRUE;
    ELSE
        P3_Pracovisko.OUT.Majak_CerveneSvetlo:= FALSE;
    END_IF

    //Zvuková signalizácia//
    //    IF EDGEPOS(P3_Pracovisko.STAV.PORUCHA) THEN
    //        P3_Pracovisko.OUT.Majak_Hukacka:= Blikac500ms;
    //    END_IF

    IF P34_AlarmyVizu.PotvrdAlarmy THEN
        P3_Pracovisko.OUT.Majak_Hukacka:= FALSE;
    END_IF

END_PROGRAM

PROGRAM _EXIT
	(* Insert code here *)

END_PROGRAM
```

#### OvlVentilovychTerminalov.st
```iecst
ACTION OvlVentilovychTerminalov:

		//Mapovanie ventilového terminálu - VT6//
	P3_Pracovisko.OUT.VT6_OUT1.0:= P3_StoperSrobovania.OUT.ZasunStoper_YV132;
	P3_Pracovisko.OUT.VT6_OUT1.1:= P3_AkumulacnyStoper.OUT.ZasunStoper_YV133;
	P3_Pracovisko.OUT.VT6_OUT1.2:= P3_LeakageTestA.OUT.ZasunStoper_YV134;
	P3_Pracovisko.OUT.VT6_OUT1.3:= P3_LeakageTestB.OUT.ZasunStoper_YV135;
	P3_Pracovisko.OUT.VT6_OUT1.4:= P3_SpodnyStoper.OUT.ZasunStoper_YV136;
	P3_Pracovisko.OUT.VT6_OUT1.5:= P3_Srobovanie.OUT.ZasobSrobK40_Ofuk_RUN_YV114;
	P3_Pracovisko.OUT.VT6_OUT1.6:= P3_Srobovanie.OUT.NastrelSrobK40_NastrelSrob_YV117;
	P3_Pracovisko.OUT.VT6_OUT1.7:= P3_Srobovanie.OUT.ZasobSrobK40_OfukTried_RUN_YV115;

	P3_Pracovisko.OUT.VT6_OUT2.0:= P3_Srobovanie.OUT.NastrelSrobK40_PosunSrobu_YV116;
	P3_Pracovisko.OUT.VT6_OUT2.1;
	P3_Pracovisko.OUT.VT6_OUT2.2:= P3_Srobovanie.OUT.SkrutkK40_PrisavSkrut_RUN_YV120;
	P3_Pracovisko.OUT.VT6_OUT2.3:= P3_Srobovanie.OUT.SkrutkK40_OfukVakua_RUN_YV119;
	P3_Pracovisko.OUT.VT6_OUT2.4:= P3_Srobovanie.OUT.SkrutkK40_Cist_OTVOR_YV121;
	P3_Pracovisko.OUT.VT6_OUT2.5;
	P3_Pracovisko.OUT.VT6_OUT2.6:= P3_Srobovanie.OUT.SkrutkK40_Cist_POSUN_YV124;
	P3_Pracovisko.OUT.VT6_OUT2.7:= P3_Srobovanie.OUT.SkrutkK40_Cist_ODSAVANIE_YV122;

	P3_Pracovisko.OUT.VT6_OUT3.0:= P3_Srobovanie.OUT.ZasobSrobM5_Ofuk_RUN_YV125;
	P3_Pracovisko.OUT.VT6_OUT3.1:= P3_Srobovanie.OUT.ZasobSrobM5_OfukTried_RUN_YV126;
	P3_Pracovisko.OUT.VT6_OUT3.2:= P3_Srobovanie.OUT.OddelovacSrobM5_OtocVZAD_YV127;
	P3_Pracovisko.OUT.VT6_OUT3.3:= P3_Srobovanie.OUT.OddelovacSrobM5_OtocVPRED_YV128;
	P3_Pracovisko.OUT.VT6_OUT3.4:= P3_Srobovanie.OUT.HVTest_PritlacKontTestera_YV140;
	P3_Pracovisko.OUT.VT6_OUT3.5:= P3_VstupnyStoper.OUT.ZasunStoper_YV193;
	P3_Pracovisko.OUT.VT6_OUT3.6:= P3_Srobovanie.OUT.SkrutkM5_PrisavSkrut_ZAPNI_YV130;
	P3_Pracovisko.OUT.VT6_OUT3.7:= P3_Srobovanie.OUT.SkrutkM5_PrisavSkrut_VYPNI_YV131;

	P3_Pracovisko.OUT.VT6_OUT4.0;
	P3_Pracovisko.OUT.VT6_OUT4.1;
	P3_Pracovisko.OUT.VT6_OUT4.2;
	P3_Pracovisko.OUT.VT6_OUT4.3;
	P3_Pracovisko.OUT.VT6_OUT4.4;
	P3_Pracovisko.OUT.VT6_OUT4.5;
	P3_Pracovisko.OUT.VT6_OUT4.6;
	P3_Pracovisko.OUT.VT6_OUT4.7;

	//Mapovanie ventilového terminálu - VT7//
	P3_Pracovisko.OUT.VT7_OUT1.0:= P3_Srobovanie.OUT.SkrutkK40_VYSUN_YV118;
	P3_Pracovisko.OUT.VT7_OUT1.1;
	P3_Pracovisko.OUT.VT7_OUT1.2:= P3_Srobovanie.OUT.SkrutkM5_VYSUN_YV129;
	P3_Pracovisko.OUT.VT7_OUT1.3;
	P3_Pracovisko.OUT.VT7_OUT1.4:= P3_StoperSrobovania.OUT.VysunCentrovanie_YV151;
	P3_Pracovisko.OUT.VT7_OUT1.5:= P3_StoperSrobovania.OUT.ZasunCentrovanie_YV152;
	P3_Pracovisko.OUT.VT7_OUT1.6:= P3_Srobovanie.OUT.HVTest_Kontakty_VYSUN_YV154;
	P3_Pracovisko.OUT.VT7_OUT1.7:= P3_Srobovanie.OUT.HVTest_Kontakty_ZASUN_YV153;

	P3_Pracovisko.OUT.VT7_OUT2.0:= P3_Srobovanie.OUT.HVTest_VYSUN_YV150;
	P3_Pracovisko.OUT.VT7_OUT2.1:= P3_Srobovanie.OUT.HVTest_ZASUN_YV149;
	P3_Pracovisko.OUT.VT7_OUT2.2:= P3_Srobovanie.OUT.HVTest_PneuPruzinu_VYSUN_YV156;
	P3_Pracovisko.OUT.VT7_OUT2.3:= P3_Srobovanie.OUT.HVTest_PneuPruzinu_ZASUN_YV155;
	P3_Pracovisko.OUT.VT7_OUT2.4:= P3_LeakageTestA.OUT.VysunCentrovanie_YV143;
	P3_Pracovisko.OUT.VT7_OUT2.5:= P3_LeakageTestA.OUT.ZasunCentrovanie_YV144;
	P3_Pracovisko.OUT.VT7_OUT2.6:= P3_LeakageTestA.OUT.Kopito_VYSUN_YV141;
	P3_Pracovisko.OUT.VT7_OUT2.7:= P3_LeakageTestA.OUT.Kopito_ZASUN_YV142;

	P3_Pracovisko.OUT.VT7_OUT3.0:= P3_LeakageTestB.OUT.VysunCentrovanie_YV147;
	P3_Pracovisko.OUT.VT7_OUT3.1:= P3_LeakageTestB.OUT.ZasunCentrovanie_YV148;
	P3_Pracovisko.OUT.VT7_OUT3.2:= P3_LeakageTestB.OUT.Kopito_VYSUN_YV145;
	P3_Pracovisko.OUT.VT7_OUT3.3:= P3_LeakageTestB.OUT.Kopito_ZASUN_YV146;
	P3_Pracovisko.OUT.VT7_OUT3.4:= P3_LeakageTestA.OUT.Pritlak_VYSUN_YV157;
	P3_Pracovisko.OUT.VT7_OUT3.5:= P3_LeakageTestA.OUT.Pritlak_ZASUN_YV158;
	P3_Pracovisko.OUT.VT7_OUT3.6:= P3_LeakageTestA.OUT.PneuZamok_ODOMKNI_YV159;
	P3_Pracovisko.OUT.VT7_OUT3.7;

	P3_Pracovisko.OUT.VT7_OUT4.0:= P3_LeakageTestB.OUT.Pritlak_VYSUN_YV161;
	P3_Pracovisko.OUT.VT7_OUT4.1:= P3_LeakageTestB.OUT.Pritlak_ZASUN_YV162;
	P3_Pracovisko.OUT.VT7_OUT4.2:= P3_LeakageTestB.OUT.PneuZamok_ODOMKNI_YV160;
	P3_Pracovisko.OUT.VT7_OUT4.3;
	P3_Pracovisko.OUT.VT7_OUT4.4;
	P3_Pracovisko.OUT.VT7_OUT4.5;
	P3_Pracovisko.OUT.VT7_OUT4.6;
	P3_Pracovisko.OUT.VT7_OUT4.7;

END_ACTION
```

#### ProfinetKomunikaciaKAM13.st
```iecst
ACTION ProfinetKomunikaciaKAM13:

	//Vstupy pre kameru//
	CAM13.Profinet_PLC_OUTPUTS[0].3:= CAM13.CMD.Triger;

	//Výstupy z kamery//
	CAM13.STAV.READY:= CAM13.Profinet_PLC_INPUTS[0].0;
	CAM13.STAV.SWITCH:= CAM13.Profinet_PLC_INPUTS[0].1;
    CAM13.STAV.BUSY:= CAM13.Profinet_PLC_INPUTS[0].2;
    CAM13.STAV.Command_AKCEPTOVANY:= CAM13.Profinet_PLC_INPUTS[0].3;
    CAM13.STAV.Command_READY:= CAM13.Profinet_PLC_INPUTS[0].4;
    CAM13.STAV.Command_ERROR:= CAM13.Profinet_PLC_INPUTS[0].5;

	//Výsledky kamery//
	CAM13.RESULT.Pritomn_SkrutkyK40_TopCover_4F5F:= CAM13.Profinet_PLC_INPUTS[2].0;
	CAM13.RESULT.Pritomn_SkrutkyM5_TopCover:= CAM13.Profinet_PLC_INPUTS[2].1;

	//Stav výsledky READY//
	IF EDGE(CAM13.STAV.SWITCH)THEN
		CAM13.STAV.Results_READY:= TRUE;
	END_IF

END_ACTION
```

### Program Logical/Program/Pracovisko_3/P3_Dopravniky (IEC)

#### Main.st - Init, cyclic, exit code
```iecst
PROGRAM _INIT
	(* Insert code here *)

END_PROGRAM

PROGRAM _CYCLIC

	//Volanie funkcie SequenceControl//
	SequenceControl(SC:= SC_P3_Dopravniky);

	//Reset sekcie //
    IF NOT Safety.STAV.P3_ZonaBunky_AKTIVNA THEN
        SC_P3_Dopravniky.Step:= 0;
    ELSIF P3_Dopravniky.Reset THEN
		SC_P3_Dopravniky.Step:= 0;
		P3_Dopravniky.Reset:= FALSE;
	END_IF

	CASE SC_P3_Dopravniky.Step OF

		0:
			SC_P3_Dopravniky.StepName:='0 - Nulovanie';
			P3_Dopravniky.Automat:= FALSE;
			P3_Dopravniky.KoniecCyklu:= FALSE;
			P3_Dopravniky.Manual:= FALSE;
			P3_Dopravniky.STAV.PoINIT:= FALSE;
			P3_Dopravniky.OUT.HornyDoprav_ChodVPRED_M33:= FALSE;
			P3_Dopravniky.OUT.SpodnyDoprav_ChodVPRED_M34:= FALSE;

			IF Safety.STAV.P3_ZonaBunky_AKTIVNA AND NOT P3_Pracovisko.STAV.PORUCHA  AND P3_Pracovisko.IN.PrivodVzduchu_SnimacTlaku_S25 THEN
				SC_P3_Dopravniky.ResetStep:= TRUE;
				SC_P3_Dopravniky.Step:= 1;
			END_IF

		1:
			SC_P3_Dopravniky.StepName:='1 - Cakam na spustenie vyroby';
			P3_Dopravniky.KoniecCyklu:= FALSE;
            IF P3_Dopravniky.Automat THEN
				SC_P3_Dopravniky.Step:= 2;
			ELSIF P3_Dopravniky.Manual THEN
				SC_P3_Dopravniky.Step:= 700;
			END_IF

			//********************************************************Inicializácia****************************************************************************//

		2:
			SC_P3_Dopravniky.StepName:='2 - Inicializacia - cakam na spustenie inicializacie';
			SC_P3_Dopravniky.IdleTime.PT:= T#2s;
			SC_P3_Dopravniky.AlarmTime.PT:= T#5s;

			IF P3_Srobovacky_VychodziaPozicia AND P3_LeakageTestA_VychodziaPozicia AND P3_LeakageTestB_VychodziaPozicia THEN
				SC_P3_Dopravniky.IdleTime.IN:= TRUE;
			ELSE
				SC_P3_Dopravniky.IdleTime.IN:= FALSE;
			END_IF

			IF SC_P3_Dopravniky.IdleTime.Q THEN
				SC_P3_Dopravniky.ResetStep:= TRUE;
				SC_P3_Dopravniky.Step:= 3;
			END_IF

		3:
			SC_P3_Dopravniky.StepName:='2 - Inicializacia - ukoncenie inicializacie';
			SC_P3_Dopravniky.IdleTime.PT:= T#4s;
			SC_P3_Dopravniky.AlarmTime.PT:= T#5s;

			P3_Dopravniky.OUT.HornyDoprav_ChodVPRED_M33:= TRUE;
			P3_Dopravniky.OUT.SpodnyDoprav_ChodVPRED_M34:= TRUE;
			SC_P3_Dopravniky.IdleTime.IN:= TRUE;

			IF SC_P3_Dopravniky.IdleTime.Q THEN
				P3_Dopravniky.STAV.PoINIT:= TRUE;
				SC_P3_Dopravniky.ResetStep:= TRUE;
				SC_P3_Dopravniky.Step:= 100;
			END_IF

			//********************************************************Automatický režim****************************************************************************//
		100:
			SC_P3_Dopravniky.StepName:='100 - Automaticky Rezim - cakam na vypnutie dopravnikou';
			SC_P3_Dopravniky.IdleTime.PT:= T#200ms;
			SC_P3_Dopravniky.AlarmTime.PT:= T#5s;

			IF P3_Dopravniky.KoniecCyklu AND NOT P3_StoperSrobovania.Automat AND NOT P3_LeakageTestA.Automat AND NOT P3_LeakageTestB.Automat AND Safety.STAV.P3_VstupBunky_Bariera_AKTIVNA AND Safety.STAV.P3_VystupBunky_Bariera_AKTIVNA THEN
				SC_P3_Dopravniky.ResetStep:= TRUE;
				SC_P3_Dopravniky.Step:= 0;
			END_IF

			//*******************************************************Manuálny režim*******************************************************************************//
		700:
			SC_P3_Dopravniky.StepName:='700 - Manualny Rezim';
			SC_P3_Dopravniky.IdleTime.PT:= T#8s;
			SC_P3_Dopravniky.AlarmTime.PT:= T#5s;

	END_CASE

END_PROGRAM

PROGRAM _EXIT
	(* Insert code here *)

END_PROGRAM
```

### Program Logical/Program/Pracovisko_3/P3_SpodnyStoper (IEC)
